FUNCTION "GCS7_SecCtrlMainMalting" : VOID	// FC 1060
TITLE = Section Control: Main function
//COPYRIGHT:    (C) 1994 BY  BUHLER AG,  CH-9240 UZWIL  SWITZERLAND
//
//PRODUCT:      GCS7
//
//TITLE:        SECTION CONTROL: MAIN PROGRAM
//
//-------------------------------------------------------------------------
//
//IDENT:        AUTOR:              DEPT:                         DATE:
//
//FC1060.1.0    M.Wedler            AEB31                         03-Feb-2005
//              Add. Code 1000 for Malting Plant only              
//FB60.3.5      A.Egli              CT3                           12-Nov-2003
//              Transition to Active: Set JobAc.BatchNo=1 when < 0
//FB60.3.4      A.Egli              CT3                           04-Aug-2003
//              PCRead.Status.StaImmediateStopASW is DBX120.0
//FB60.3.3      A.Egli              CT3                           17-Jul-2003
//              PCDirectControl: ParLineNr is DBW2 and not DBW4
//FB60.3.2      A.Egli              CT3                           12-Jun-2003
//              Wrong lenght copy Line to section
//FB60.3.1      A.Egli              CT3                           14-Mar-2003
//              Code35: Move to any section DB: DBW20=Destination
//              Code22,23: No Transition StEmptying to StWait
//FB60.3.0      A.Egli              CT3                            8-Okt-2002
//              New release
//FB60.2.10     A.Egli              CT3                           18-Mar-2002
//  Send Command only to next section, if InfDataReady=1
//FB60.2.9      A.Egli              CT3                           24-Sept-2001
//  ParStartReleaseTime <=0 : Unlimited time
//FB60.2.8      A.Egli              CT3                           17-Mai-2001
//  Update Last Batch in next section
//FB60.2.7      A.Egli              CT3                            5-Jul-2000
//  Read command from PC only with F_Define 
//FB60.2.6      A.Egli              CT3                           13-Mar-2000
//  Replace DBB73 with DBW72 and DBB9 with DBW8 
//FB60.2E       A.Egli              CT3                           30-Apr-1999
// -Zustandswechsel nach st_emptied: Abfrage DBX117.3 nicht DIX117.3 
//FB60.2D       A.Egli              CT3                           01-Apr-1999
// -Methode 25: Move allways
// -Bei reset Zustandswechsel nach st_emptied (Verbuchung
// -Bei reset kein Zustandswechsel nach  StActive
//FB60.2C       A.Egli              CT3                           22-Jul-98
//               Line-Nr =DBW2
//FB60.2B       A.Egli              AEE6                          14-Mai-98
//               ToASW.InfDataMoved
//FB60.2A       A.Egli              AEE6                          14-Jan-98
//               Update  S5 (Version 2M)
//FB60.1A       A.Egli              AEE6                          16-Jun-96
//               Convert S5 to S7 (Version 2H)
//
//-------------------------------------------------------------------------
//
//PURPOSE:      MANUAL : GCSOSMAN
//
//RESTRICTIONS:
//
//-------------------------------------------------------------------------
//
// CODE of the Methode
//        0    : METHODE CONTROL
//        1    : METHODE DECODER
//        2    : METHODE STEP
//        3    : METHODE STEP_TRANSITION
//        4    : METHODE STATE
//        5    : METHODE MOVE_DATA
//        6    : METHODE NEXT BATCH
//        7    : METHODE O_SECTION
//        9    : METHODE ResultTotal
//        10   : METHODE ResultBatch
//        12   : METHODE PC Direct Control (Diagnose)
//        13   : METHODE WayAdJustTime  
//        25   : METHODE MOVE_DATA Uncondtion
//        35   : METHODE MOVE_DATA any section
//
//ACTUAL DB BY CALL: SECTION  DB
//AUFGESCHALGENER  : SEKTIONS DB
//
//$EJECT
//
//
//
//
//
AUTHOR : EA
FAMILY : GCS7UL
NAME : SEC_MAIN
VERSION : 3.5
VAR_INPUT
  CODE : INT ;	// CODE
END_VAR
VAR_TEMP
  Fault : BOOL ;
  VarLength : INT ;
  tmpByteWrite : INT ;
  SecDBAc : INT ;
  SecDBNext : INT ;
END_VAR
BEGIN
NETWORK
TITLE =
      L     DBNO;
      T     #SecDBAc;
NETWORK
TITLE =  METHODE CONTROL
//Functions :
// - Section Commands 
//   > Sec.ToSSW.Func (commands last cycle) or'd with ToASW.Func
//   > Sec.ToASW.Func (commands) partially processed
// - Section Emptying Time controlled
// - Section F_Result controlled
//
//Called by : Section FC
      L     #CODE;
      L     0;	// METHODE CONTROL
      <>I;	// with Check JOB and Batch Status
      A(;
      L     #CODE;
      L     1000;	// METHODE CONTROL
      <>I;	// without Check JOB and Batch Status
      );
      JC    aEnd;
// === COMMANDS =====================================
      L     DBD 46;	// "SecDB".ToASW.Func
      L     DBD 66;	// "SecDB".ToSSW.Func
      OD;	// 
      T     DBD 46;	//>"SecDB".ToASW.Func
      L     0;	// 
      ==D;	// no new commands
      JC    aNoC;
// --- RESET STATUSBIT -----
      L     2#111111;	// ON-COMMAND
      L     DBW 46;	// "SecDB".ToASW.Func[31..16]
      AW;	// 
      INVI;	// 
      L     DBW 120;	// "SecDB".PCRead.Status[15..00]
      AW;	// 
      T     DBW 120;	//>"SecDB".PCRead.Status[15..00]
// --- SET STATUSBIT  ------
      L     2#11111111;	// OFF-COMMAND
      L     DBW 48;	// "SecDB".ToASW.Func[15..00]
      AW;	// 
      L     DBW 120;	// "SecDB".PCRead.Status[15..00]
      OW;	// 
      T     DBW 120;	//>"SecDB".PCRead.Status[15..00]
// 
// M.W. 03.02.05 
      L     #CODE;
      L     1000;	// METHODE CONTROL
      ==I;	// without Check JOB and Batch Status
      JC    nRes;
      JU    res;
nRes: NOP   0;
      R     DBX 48.1;	// "SecDB".ToASW.Func.CmdAbortBatch
      R     DBX 49.6;	// "SecDB".ToASW.Func.CmdReset
      R     DBX 49.7;	// "SecDB".ToASW.Func.CmdSequenzStop
//      R     DBX  121.0                  // "SecDB".PCRead.Status.StaImediateStop
      R     DBX 121.6;	// "SecDB".PCRead.Status.StaReset
      R     DBX 121.7;	//>"SecDB".PCRead.Status.StaEndOfJob
res:  NOP   0;
// 
      A     DBX 121.6;	// "SecDB".PCRead.Status.StaReset
      S     DBX 121.7;	//>"SecDB".PCRead.Status.StaEndOfJob
      A     DBX 48.1;	// "SecDB".ToASW.Func.CmdAbortBatch
      S     DBX 201.0;	//>"SecDB".JobAc.StaBatch.StaErrBatch
      A     DBX 49.6;	// "SecDB".ToASW.Func.CmdReset
      O     DBX 49.7;	// "SecDB".ToASW.Func.CmdSequenzStop
      O     DBX 48.1;	// "SecDB".ToASW.Func.CmdAbortBatch
      A     DBX 45.7;	// "SecDB".ToASW.InfDataReady [2.10]
      JCN   aNoC;
      CALL  "GCS7_SecCtrlSubMalting" (
           CODE                     := 2);	// SUBROUTINE sequenz_stop (Code 2)
aNoC: L     0;	// 
      T     DBD 66;	//>"SecDB".ToSSW.Func
      L     DBW 206;	// "SecDB".JobAc.BatchNo
      L     DBW 168;	// "SecDB".JobNom.BatchNo
      >=I;	// 
      S     DBX 201.3;	//>"SecDB".JobAc.StaBatch.StaLastBatch
// M.W.
      L     #CODE;
      L     1000;	// METHODE CONTROL
// M.W. 04.10.04
//      <>I                               // without Check JOB and Batch Status
      ==I;
      JC    aETI;	// -> Emptying Time
      CALL  "GCS7_SecCtrlSubMalting" (
           CODE                     := 1);	// SUBROUTINE compare (Code 1)
// === EMPTYING TIME ==================================
aETI: NOP   0;
      AN    DBX 64.2;	// "SecDB".ToSSW.InfPulseTimer
      O     DBX 45.0;	// "SecDB".ToASW.InfEmptyingTimeEnd
      JC    aE2;	// 
      L     DBW 132;	// "SecDB".PCRead.OutEmptyingTime
      +     1;	// 
      T     DBW 132;	//>"SecDB".PCRead.OutEmptyingTime
// 
aE2:  A     DBX 62.5;	// "SecDB".ToSSW.InfFeeding
      S     DBX 119.4;	//>"SecDB".PCRead.Status.StaLoaded
      A     DBX 64.7;	// "SecDB".ToSSW.InfReleaseEmptyingTime
      JC    aX3;	// 
      L     0;	// 
      T     DBW 132;	//>"SecDB".PCRead.OutEmptyingTime
aX3:  L     DBW 100;	// "SecDB".PCWrite.ParEmptyingTime
      L     DBW 132;	// "SecDB".PCRead.OutEmptyingTime
      <=I;	// 
      A     DBX 64.7;	// "SecDB".ToSSW.InfReleaseEmptyingTime 
      =     DBX 45.0;	// "SecDB".ToASW.InfEmptyingTimeEnd
      R     DBX 119.4;	//>"SecDB".PCRead.Status.StaLoaded
      AN    DBX 45.0;	// "SecDB".ToASW.InfEmptyingTimeEnd
      A     DBX 64.7;	// "SecDB".ToSSW.InfReleaseEmptyingTime
      =     DBX 119.6;	//>"SecDB".PCRead.Status.StaEmptyingTime
// === F_RESULT ========================================
      AN    DBX 64.1;	// "SecDB".ToSSW.CmdSendResult
      JC    aCMD;	// 
      AN    DBX 82.1;	// "SecDB".PCWrite.Hsk.Q_Result
      AN    DBX 201.2;	// "SecDB".JobAc.StaBatch.StaRegistrated
      AN    DBX 102.1;	// "SecDB".PCRead.Hsk.F_Result
      S     DBX 102.1;	//>"SecDB".PCRead.Hsk.F_Result
      S     DBX 41.0;	//>"SecDB".ChangeBit.CBit1 
aCMD: BEU;
aEnd: NOP   0;
NETWORK
TITLE =  METHODE DECODER (Code 1)
//Functions :
// -Copies Job data (obj64) from L_DB to all S_DB with the same job.
// -Calls initialise for sections with new job (F_Execute)
//
//Called by : Line FC
//Special : LCTRLMAIN INIT(1) must be called before this function
      L     #CODE;
      L     1;	// METHODE DECODER
      <>I;
      JC    bEnd;
      L     0;
      L     DBB 145;	// "LineDB".JobWrite.Hsk
      ==I;
      BEC;
      L     DBW 140;	// "LineDB".JobRead.ErrCode   [*1C*]
      L     0;
      <>I;
      BEC;
      L     64;	// Job Header
      T     DBW 20;	//>"LineDB".VarTemp[1] = ObjectNr
      CALL  FC 59 (
           $1                       := 1);	// SUBROUTINE Object Address (code 1)
      OPN   DI [DBW 4];	// >>> FIRST SECTION-DB[ "LineDB".Para.ParFirstSecDB]
bLop: AN    DIX 44.7;	// "SecDB".ToASW.InfSameJobLineDB
      JC    bNxt;
// === COMMANDS ========================================
      S     DIX 44.0;	//>"SecDB".ToASW.CmdModify  
      L     DBD 156;	// "LineDB".JobWrite.Func
      L     DID 46;	// "SecDB".ToASW.Func
      OD;	// 
      T     DID 46;	//>"SecDB".ToASW.Func
// === COPY JOB-HEADER (JObNom)=========================
      L     DINO;
      T     #SecDBAc;
      CALL  FC 49 (
           $1                       := P#DIX 4.0,
           $2                       := 160,
           $3                       := #SecDBAc,
           $4                       := 160,
           $5                       := 40,
           $6                       := #Fault);	// L_DB /  L_DB.JobNom /  S_DB /  S_DB.JobNom /  JobNom
// === COPY ADDITIONAL DATA (SecNom)====================
      L     DBW 22;	// "LineDB".VarTemp[2]= VarDWNr
      L     0;	// 
      ==I;	// 
      JC    bEXE;	// 
      L     DIW 12;	// "SecDB".Para.ParSecDataLenNomValue
      T     #VarLength;	//>VarLength
      L     DIW 10;	// "SecDB".Para.ParSecDataFirstByte
      L     DIW 14;	// "SecDB".Para.ParSecDataLenAcValue [3.1]
      +I;
      T     #tmpByteWrite;
      CALL  FC 49 (
           $1                       := P#DIX 4.0,
           $2                       := P#DBX 22.0,
           $3                       := #SecDBAc,
           $4                       := #tmpByteWrite,
           $5                       := #VarLength,
           $6                       := #Fault);	// L_DB /  L_DB.VarDWNr /  S_DB
bEXE: AN    DBX 145.1;	// "LineDB".JobWrite.Hsk.F_Execute
      JC    bNxt;
      R     DBX 153.7;	//>"LineDB".JobWrite.ObjMask[64]
      L     DBD 146;	// "LineDB".JobWrite.ObjMask[64..01]
      L     DBD 150;	// "LineDB".JobWrite.ObjMask[64..01]
      OD;
      JN    bNxt;
      CDB;
      CALL  "GCS7_SecCtrlSubMalting" (
           CODE                     := 3);	// SUBROUTINE init_section
      CDB;
// -- Call next section
bNxt: L     DIW 8;	// "SecDB".Para.ParNextSecDB
      L     0;	//  
      ==I;	// no next section
      JC    bINI;	// 
      OPN   DI [DIW 8];	//>>> NEXT SECTION-DB["SecDB".Para.ParNextSecDB]
      JU    bLop;
bINI: R     DBX 153.7;	//>"LineDB".JobWrite.ObjMask[64]
      BEU;
bEnd: NOP   0;
NETWORK
TITLE =  METHODE STEP (Code 2 , 22) 
//Functions :
// - Tests for step transitions from current step "SecDB".PCRead.Step
//   > Output SecDB".ToASW.Transition 
//
//Called by : Section FC
      L     #CODE;
      L     2;	// METHODE STEP
      <>I;
      A(;
      L     #CODE;
      L     22;
      <>I;
      );
      JC    cEnd;
      L     0;
      T     DBW 50;	// "SecDB".ToASW.Transition:=0
      A     DBX 111.0;	// "SecDB".PCRead.Step.StPassive
      JC    cS0;
      A     DBX 111.1;	// "SecDB".PCRead.Step.StWait
      JC    cS1;	// 
      A     DBX 111.2;	// "SecDB".PCRead.Step.StActive
      JC    cS2;
      A     DBX 111.3;	// "SecDB".PCRead.Step.StReady
      JC    cS3;
      A     DBX 111.4;	// "SecDB".PCRead.Step.StEmptying
      JC    cS4;
      A     DBX 111.5;	// "SecDB".PCRead.Step.StEmptied
      JC    cS5;
      A     DBX 111.6;	// "SecDB".PCRead.Step.StIdling
      JC    cS6;
      S     DBX 111.0;	// "SecDB".PCRead.Step.StPassive
// === "SecDB".PCRead.Step.StPassive ===================
cS0:  A     DBX 45.7;	// "SecDB".ToASW.InfDataReady
      JC    cTx1;	//>Transition.ToWait
      JU    cEnd;
// === "SecDB".PCRead.Step.StWait ======================
cS1:  A(;
      L     #CODE;
      L     2;
      ==I;
      );
      A     DBX 121.7;	// "SecDB".PCRead.Status.StaEndOfJob
      AN    DBX 44.5;	// "SecDB".ToASW.InfSameBatchPrevSec
      O     DBX 121.6;	// "SecDB".PCRead.Status.StaReset
      ON    DBX 45.7;	// "SecDB".ToASW.InfDataReady
      JC    cTx5;	//>Transition.ToEmptied [2D]
      AN    DBX 116.0;	// "SecDB".PCRead.fault.EsBatchSize
      A     DBX 63.1;	// "SecDB".ToSSW.CmdGotoActive
      JC    cTx2;	//>Transition.ToActive
      JU    cEnd;
// === "SecDB".PCRead.Step.StActive ====================
cS2:  A     DBX 63.2;	// "SecDB".ToSSW.CmdGotoReady
      AN    DBX 44.5;	// "SecDB".ToASW.InfSameBatchPrevSec
      JC    cTx3;	//>Transition.ToReady
      L     DBW 72;	// "SecDB".ToSSW.InNextSecDB
      L     0;	// 
      ==I;	// 
      O     DBX 44.6;	// "SecDB".ToASW.InfSameBatchNextSec
      AN    DBX 44.5;	// "SecDB".ToASW.InfSameBatchPrevSec
      A     DBX 63.3;	// "SecDB".ToSSW.CmdGotoEmptying
      JC    cTx4;	//>Transition.ToEmptying 
      A     DBX 121.6;	// "SecDB".PCRead.Status.StaReset
      ON    DBX 45.7;	// "SecDB".ToASW.InfDataReady
      JC    cTx5;	//>Transition.ToEmptied [2D]
      JU    cEnd;
// ===  "SecDB".PCRead.Step.StReady ====================
cS3:  L     DBW 72;	// "SecDB".ToSSW.InNextSecDB
      L     0;	// 
      ==I;	// 
      O     DBX 44.6;	// "SecDB".ToASW.InfSameBatchNextSec
      A     DBX 63.3;	// "SecDB".ToSSW.CmdGotoEmptying
      JC    cTx4;	//>Transition.ToEmptying 
      A     DBX 121.6;	// "SecDB".PCRead.Status.StaReset
      ON    DBX 45.7;	// "SecDB".ToASW.InfDataReady
      JC    cTx5;	//>Transition.ToEmptied [2D]
      JU    cEnd;
// === "SecDB".PCRead.Step.StEmptying ===================
cS4:  A     DBX 44.5;	// "SecDB".ToASW.InfSameBatchPrevSec
      JC    cTx2;	//>Transition.ToActive
      L     DBW 72;	// "SecDB".ToSSW.InNextSecDB
      L     0;	// 
      ==I;	// 
      O     DBX 44.6;	// "SecDB".ToASW.InfSameBatchNextSec
      A     DBX 63.4;	// "SecDB".ToSSW.CmdGotoEmptied
      JC    cTx5;	//>Transition.ToEmptied
      A     DBX 121.6;	// "SecDB".PCRead.Status.StaReset
      ON    DBX 45.7;	// "SecDB".ToASW.InfDataReady 
      JC    cTx5;	//>Transition.ToEmptied [2D]
      JU    cEnd;
// === "SecDB".PCRead.Step.StEmptied=====================
cS5:  A     DBX 44.5;	// "SecDB".ToASW.InfSameBatchPrevSec
      AN    DBX 121.6;	// "SecDB".PCRead.Status.StaReset [2D]
      JC    cTx2;	//>Transition.ToActive
      L     DBW 206;	// "SecDB".JobAc.BatchNo 
      L     DBW 168;	// "SecDB".JobNom.BatchNo
      >=I;	// 
      S     DBX 121.7;	//>"SecDB".PCRead.Status.StaEndOfJob
      L     0;	// 
      L     DBW 70;	// "SecDB".ToSSW.InPrevSecDB
      ==I;	// 
      A(;
      L     #CODE;
      L     22;
      <>I;
      );
      AN    DBX 121.6;	// "SecDB".PCRead.Status.StaReset 
      AN    DBX 121.7;	// "SecDB".PCRead.Status.StaEndOfJob
      A     DBX 45.7;	// "SecDB".ToASW.InfDataReady
      A     DBX 63.5;	// "SecDB".ToSSW.CmdGotoIdling
      JC    cTx1;	//>Transition.ToWait
      A     DBX 121.6;	// "SecDB".PCRead.Status.StaReset [2D]
      ON    DBX 45.7;	// "SecDB".ToASW.InfDataReady
      AN    DBX 119.3;	// "SecDB".PCRead.Status.StaOnline [2E]
      O     DBX 63.5;	// "SecDB".ToSSW.CmdGotoIdling
      JC    cTx6;	//>Transition.ToIdling
      JU    cEnd;
// === "SecDB".PCRead.Step.StIdling =====================
cS6:  A     DBX 45.7;	// "SecDB".ToASW.InfDataReady
      JC    cTx1;	//>Transition.ToWait
      A     DBX 63.6;	// "SecDB".ToSSW.CmdGotoPassive
      JC    cTx0;	//>Transition.ToPassive
      JU    cEnd;
// === SET TRANSITION ===================================
cTx0: L     2#1;	// "SecDB".ToASW.Transition.ToPassive
      JU    cTra;	// 
cTx1: L     2#10;	// "SecDB".ToASW.Transition.ToWait
      JU    cTra;	// 
cTx2: L     2#100;	// "SecDB".ToASW.Transition.ToActive
      JU    cTra;	// 
cTx3: L     2#1000;	// "SecDB".ToASW.Transition.ToReady
      JU    cTra;	// 
cTx4: L     2#10000;	// "SecDB".ToASW.Transition.ToEmptying
      JU    cTra;	// 
cTx5: L     2#100000;	// "SecDB".ToASW.Transition.ToEmptied
      JU    cTra;	// 
cTx6: L     2#1000000;	// "SecDB".ToASW.Transition.ToIdling
// ==== WRITE TRANSITION ================================
cTra: T     DBW 50;	//>"SecDB".ToASW.Transition
      BEU;
cEnd: NOP   0;
NETWORK
TITLE =  METHODE TRANSITION_STEP (code 3)
//Functions :
// - Manages Step Transitions "SecDB".ToASW.Transition
//   > Writes transition specific commands
//   > Output SecDB".ToASW.Step
//
//Called by : Section FC
      L     #CODE;
      L     3;	// METHODE TRANSITION STEP 
      <>I;
      A(;
      L     #CODE;
      L     23;
      <>I;
      );
      JC    dEnd;
      L     DBW 50;	// "SecDB".ToASW.Transition
      L     0;	// 
      ==I;	// 
      BEC;	// EXIT
      A     DBX 51.0;	// "SecDB".ToASW.Transition.ToPassive
      JC    dTx0;
      A     DBX 51.1;	// "SecDB".ToASW.Transition.ToWait
      JC    dTx1;
      A     DBX 51.2;	// "SecDB".ToASW.Transition.ToActive 
      JC    dTx2;
      A     DBX 51.3;	// "SecDB".ToASW.Transition.ToReady
      JC    dTx3;
      A     DBX 51.4;	// "SecDB".ToASW.Transition.ToEmptying
      JC    dTx4;
      A     DBX 51.5;	// "SecDB".ToASW.Transition.ToEmptied 
      JC    dTx5;
      A     DBX 51.6;	// "SecDB".ToASW.Transition.ToIdling
      JC    dTx6;
      JU    dEnd;
// === "SecDB".ToASW.Transition.ToPassive ===============
dTx0: NOP   0;
      JU    dTra;
// === "SecDB".ToASW.Transition.ToWait ==================
dTx1: R     DBX 63.1;	// "SecDB".ToSSW.CmdGotoActive 
      R     DBX 64.1;	// "SecDB".ToSSW.CmdSendResult
      A     DBX 111.5;	// "SecDB".PCRead.Step.StEmptied 
      R     DBX 201.0;	//>"SecDB".JobAc.StaBatch.StaErrBatch
      JU    dTra;
// === "SecDB".ToASW.Transition.ToActive ================
dTx2: R     DBX 63.2;	//>"SecDB".ToSSW.CmdGotoReady
      R     DBX 63.3;	//>"SecDB".ToSSW.CmdGotoEmptying
      R     DBX 64.1;	//>"SecDB".ToSSW.CmdSendResult
      L     DBW 206;	// "SecDB".JobAc.BatchNo  [3.5]
      L     1;	//                        [3.5]
      >=I;	//                        [3.5]
      ON    DBX 200.6;	// "SecDB".JobAc.StaBatch.StaEmptyingBatch [3.5]
      JC    dTra;	//                        [3.5]
      T     DBW 206;	// "SecDB".JobAc.BatchNo  [3.5]
      JU    dTra;
// === "SecDB".ToASW.Transition.ToReady =================
dTx3: R     DBX 63.3;	//>"SecDB".ToSSW.CmdGotoEmptying
      JU    dTra;
// === "SecDB".ToASW.Transition.ToEmptying ==============
dTx4: R     DBX 63.4;	//>"SecDB".ToSSW.CmdGotoEmptied
      JU    dTra;
// === "SecDB".ToASW.Transition.ToEmptied ===============
dTx5: R     DBX 63.5;	//>"SecDB".ToSSW.CmdGotoIdling
      JU    dTra;
// === "SecDB".ToASW.Transition.ToIdling ================
dTx6: R     DBX 63.6;	//>"SecDB".ToSSW.CmdGotoPassive
      R     DBX 201.0;	//>"SecDB".JobAc.StaBatch.StaErrBatch
      R     DBX 200.7;	//>"SecDB".JobAc.StaBatch.StaScaleRecipeValid
      AN    DBX 121.7;	// "SecDB".PCRead.Status.StaEndOfJob [2.8]
      JC    dT61;	// [2.8]                
      CALL  "GCS7_SecCtrlSubMalting" (
           CODE                     := 2);	// SUBROUTINE sequenz_stop [2.8]
dT61: L     0;	// 
      L     DBW 70;	// "SecDB".ToSSW.InPrevSecDB 
      <>I;	// 
      O(;
      L     #CODE;
      L     23;
      ==I;
      );
      O     DBX 121.7;	// "SecDB".PCRead.Status.StaEndOfJob
      R     DBX 45.7;	//>"SecDB".ToASW.InfDataReady
      CALL  "GCS7_SecCtrlSubMalting" (
           CODE                     := 7);	// Subroutine TestDone
      AN    DBX 39.0;	// OUTP.JobNotFound
      JC    dTra;	// 
      AN    DBX 102.0;	// "SecDB".PCRead.Hsk.F_Status 
      S     DBX 201.4;	//>"SecDB".JobAc.StaBatch.StaDone
      S     DBX 102.0;	//>"SecDB".PCRead.Hsk.F_Status
      S     DBX 41.0;	//>"SecDB".ChangeBit.CBit1
dTra: L     DBW 50;	// "SecDB".ToASW.Transition
      T     DBB 111;	//>"SecDB".PCRead.Step
      SET;	// 
      S     DBX 41.0;	//>"SecDB".ChangeBit.CBit1
      BEU;
dEnd: NOP   0;
NETWORK
TITLE =  METHODE STATE Code4
//Functions :
// - Processes SumState "SecDB".PCRead.State
//   > Output "SecDB".PCRead.State
//
//Called by : Section FC
      L     #CODE;
      L     4;	// METHODE STATE
      <>I;
      JC    eEnd;
      A     DBX 113.0;	// "SecDB".PCRead.State.StStopped
      JC    eS0;
      A     DBX 113.1;	// "SecDB".PCRead.State.StStarting
      JC    eS1;
      A     DBX 113.2;	// "SecDB".PCRead.State.StStarted 
      JC    eS2;
      A     DBX 113.3;	// "SecDB".PCRead.State.StStopping
      JC    eS3;
      A     DBX 113.5;	// "SecDB".PCRead.State.StFeeding
      JC    eS4;
      S     DBX 113.0;	// "SecDB".PCRead.State.StStopped
// === "SecDB".PCRead.State.StStopped ===================
eS0:  AN    DBX 62.0;	// "SecDB".ToSSW.InfStopped
      JC    eT01;	//>State.StStarting
      JU    eEnd;	// 
eT01: L     2#10;	//>"SecDB".PCRead.State.StStarting
      JU    eTra;
// === "SecDB".PCRead.State.StStarting ==================
eS1:  A     DBX 62.2;	// "SecDB".ToSSW.InfStarted
      JC    eT12;	//>State.StStarted
      A     DBX 120.0;	// "SecDB".PCRead.Status.StaImmediateStopASW // [3.4]
      O     DBX 62.0;	// "SecDB".ToSSW.InfStopped
      O     DBX 111.6;	// "SecDB".PCRead.Step.StIdling
      JC    eT13;	//>State.StStopping
      JU    eEnd;
eT12: L     2#100;	//>"SecDB".PCRead.State.StStarted
      JU    eTra;
eT13: L     2#1000;	//>"SecDB".PCRead.State.StStopping
      JU    eTra;
// === "SecDB".PCRead.State.StStarted ===================
eS2:  A     DBX 120.0;	// "SecDB".PCRead.Status.StaImmediateStopASW
      O     DBX 62.0;	// "SecDB".ToSSW.InfStopped
      JC    eT23;	//>State.StStopping
      AN    DBX 62.2;	// "SecDB".ToSSW.InfStarted
      JC    eT21;	//>State.StStarting
      A     DBX 62.5;	// "SecDB".ToSSW.InfFeeding
      JC    eT25;	//>State.StFeeding
      JU    eEnd;
eT21: L     2#10;	//>"SecDB".PCRead.State.StStarting
      JU    eTra;
eT23: L     2#1000;	//>"SecDB".PCRead.State.StStopping
      JU    eTra;
eT25: L     2#100000;	//>"SecDB".PCRead.State.StFeeding
      JU    eTra;
// === "SecDB".PCRead.State.StStopping ==================
eS3:  A     DBX 62.0;	// "SecDB".ToSSW.InfStopped
      JC    eT30;	//>State.StStopped
      AN    DBX 120.0;	// "SecDB".PCRead.Status.StaImmediateStopASW
      AN    DBX 62.0;	// "SecDB".ToSSW.InfStopped
      A     DBX 62.2;	// "SecDB".ToSSW.InfStarted
      JC    eT32;	//>State.StStarted
      AN    DBX 120.0;	// "SecDB".PCRead.Status.StaImmediateStopASW
      AN    DBX 111.6;	// "SecDB".PCRead.Step.StIdling
      JC    eT32;	//>State.StStarting
      JU    eEnd;
eT30: L     2#1;	//>"SecDB".PCRead.State.StStopped
      JU    eTra;
eT32: L     2#100;	//>"SecDB".PCRead.State.StStarted
      JU    eTra;
      L     2#10;	//>"SecDB".PCRead.State.StStarting
      JU    eTra;
// === "SecDB".PCRead.State.StFeeding ===================
eS4:  AN    DBX 62.5;	// "SecDB".ToSSW.InfFeeding
      JC    eT52;	//>State.StStarted
      JU    eEnd;	// 
eT52: L     2#100;	//>"SecDB".PCRead.State.StStarted
// ==== SET STATE (TRANSITION) ==========================
eTra: T     DBB 113;	//>"SecDB".PCRead.State
      SET;	// 
      S     DBX 41.0;	//>"SecDB".Changebit.CBit1
      BEU;
eEnd: NOP   0;
NETWORK
TITLE =  METHODE MOVE_DATA Code 5,25,35
//Function :
// - Manages Section to Section Job Copy for Job and Bin Data 
// > Code 5: Regular copy to next section
// > Code 25:Unconditional copy to next section
// > Code 35:Regular copy to specified section destination (DBW20)
// > Output : Job Ac, Job Nom, Sec Ac, Sec Nom, Bin Recipe. Copied Section to 
//Section 
//
//Called by : Section FC
      L     #CODE;
      L     5;	// METHODE MOVE DATA Next Section Regular
      ==I;
      JC    m5;
      L     #CODE;
      L     25;	// METHODE MOVE DATA Next Section Unconditional
      ==I;
      JC    m25;
      L     #CODE;
      L     35;	// METHODE MOVE DATA Any Section Regular
      <>I;
      JC    fEnd;
// === Move to section DBW20 (Code 35)===============
      R     DBX 44.2;	// S_DB[n  ].ToASW.CmdDataMoved
      L     0;
      L     DBW 20;	// S_DB[n  ].VarTemp.InOutValue1
      ==I;	// 
      BEC;	//>No next section
      T     #SecDBNext;
      OPN   DI [#SecDBNext];	// >>>CALL NEXT SECTION ["SecDB".ToSSW.InNextSecDB]
      JU    m35;	//> Regular Conditions
//====== Move Uncondition (Code=25) =================
m25:  R     DBX 44.2;	// S_DB[n  ].ToASW.CmdDataMoved
      L     DBW 72;	// S_DB[n  ].ToSSW.InNextSecDB
      L     0;	// 
      ==I;	// 
      BEC;	//>No next section
      AN    DBX 44.6;	// S_DB[n  ].ToASW.InfSameBatchNextSec
      OPN   DI [DBW 72];	// >>> NEXT SECTION ["SecDB".ToSSW.InNextSecDB]
      A     DIX 64.0;	// S_DB[n+1].ToSSW.InfReadyForNewBatch
      AN    DIX 121.3;	// S_DB[n+1].PCRead.Status.StaHold
      A(;
      AN    DIX 102.0;	// S_DB[n+1].PCRead.Hsk.F_Status
      ON    DIX 119.3;	// S_DB[n+1].PCRead.Status.StaOnline
      );
      JC    C3;	//>Move Data
      BEU;
//=== Move Regular (Code=5) =========================
m5:   R     DBX 44.2;	// S_DB[n  ].ToASW.CmdDataMoved
      A     DBX 44.6;	// S_DB[n  ].ToASW.InfSameBatchNextSec
      BEC;	//  
      L     DBW 72;	// S_DB[n  ].ToSSW.InNextSecDB
      L     0;	// 
      ==I;	// 
      BEC;	//>No next section
      OPN   DI [DBW 72];	// >>> NEXT SECTION-DB["SecDB".ToSSW.InNextSecDB]
m35:  A     DBX 201.0;	// S_DB[n  ].JobAc.StaBatch.StaErrBatch
      A     DIX 45.7;	// S_DB[n+1].ToASW.InfDataReady
      BEC;	// 
      A     DIX 165.0;	// S_DB[n+1].sta_err_batch
      A     DIX 45.7;	// S_DB[n+1].ToASW.InfDataReady
      BEC;	// 
      A     DIX 111.0;	// S_DB[n+1].PCRead.Step.StPassive
      O     DIX 111.6;	// S_DB[n+1].PCRead.Step.StIdling
      O     DIX 111.4;	// S_DB[n+1].PCRead.Step.StEmptying
      O     DIX 111.5;	// S_DB[n+1].PCRead.Step.StEmptied
      JC    C2;
      BEU;
      AN    DBX 45.7;	// S_DB[n  ].ToASW.InfDataReady
      O     DBX 44.3;	// S_DB[n  ].ToASW.InfSameJobPrevSec
      A     DBX 64.0;	// S_DB[n  ].ToSSW.InfReadyForNewBatch
      AN    DBX 121.3;	// S_DB[n  ].PCRead.Status.StaHold
      A(;
      AN    DBX 102.0;	// S_DB[n  ].PCRead.Hsk.F_Status
      ON    DBX 119.3;	// S_DB[n  ].PCRead.Status.StaOnline
      );
C2:   AN    DIX 45.7;	// S_DB[n+1].ToASW.InfDataReady
      O     DIX 44.3;	// S_DB[n+1].ToASW.InfSameJobPrevSec
      A     DIX 64.0;	// S_DB[n+1].ToSSW.InfReadyForNewBatch
      AN    DIX 121.3;	// S_DB[n+1].PCRead.Status.StaHold
      A(;
      AN    DIX 102.0;	// S_DB[n+1].PCRead.Hsk.F_Status
      ON    DIX 119.3;	// S_DB[n+1].PCRead.Status.StaOnline
      );
      JC    C3;
      BEU;
// === MOVE DATA =======================================
// --- Copy Header (JobAc + JobNom)---------------------
C3:   L     DINO;
      T     #SecDBNext;
      CALL  FC 49 (
           $1                       := #SecDBAc,
           $2                       := 160,
           $3                       := #SecDBNext,
           $4                       := 160,
           $5                       := 80,
           $6                       := #Fault);	// S_DB[n  ].JobNom /  S_DB[n+1].JobNom /  JobAc + JobNom
// --- Copy Dynamic Datas (SecAc + SecNom)--------------
      L     DIW 14;	// S_DB[n+1].Para.ParSecDataLenAcValue
      L     DIW 12;	// S_DB[n+1].Para.ParSecDataLenNomValue
      +I;
      T     #VarLength;
      CALL  FC 49 (
           $1                       := #SecDBAc,
           $2                       := P#DBX 10.0,
           $3                       := #SecDBNext,
           $4                       := P#DIX 10.0,
           $5                       := #VarLength,
           $6                       := #Fault);	// S_DB[n  ].Para.ParSecDataFirstByte /  S_DB[n+1].Para.ParSecDataFirstByte /  SecAc + SecNom
// --- Copy Bin Data (Recipe) ---------------------------
      CALL  FC 49 (
           $1                       := #SecDBAc,
           $2                       := P#DBX 16.0,
           $3                       := #SecDBNext,
           $4                       := P#DIX 16.0,
           $5                       := P#DIX 18.0,
           $6                       := #Fault);	// S_DB[n  ].Para.ParBinDataFirstByte /  S_DB[n+1].Para.ParBinDataFirstByte /  S_DB[n+1].Para.ParBinDataLength
// --- Initalise S_DB[n+1] ------------------------------
      SET;
      S     DIX 45.7;	// S_DB[n+1].ToASW.InfDataReady 
      S     DIX 44.1;	// S_DB[n+1].ToASW.CmdNewBatch
      S     DBX 44.2;	// S_DB[n  ].ToASW.CmdDataMoved
      R     DIX 121.6;	// S_DB[n+1].PCRead.Status.StaReset
      R     DIX 121.7;	// S_DB[n+1].PCRead.Status.StaEndOfJob
      R     DIX 64.1;	// S_DB[n+1].ToSSW.CmdSendResult
      AN    DBX 121.0;	// S_DB[n  ].PCRead.Status.StaImmediateStop   
      R     DIX 121.0;	// S_DB[n+1].PCRead.Status.StaImmediateStop      
      AN    DBX 121.1;	// S_DB[n  ].PCRead.Status.StaTransferOff
      R     DIX 121.1;	// S_DB[n+1].PCRead.Status.StaTransferOff
      AN    DBX 121.2;	// S_DB[n  ].PCRead.Status.StaFeedOff
      R     DIX 121.2;	// S_DB[n+1].PCRead.Status.StaFeedOff
      CDB;	// >>> DB to DI
      CALL  "GCS7_SecCtrlSubMalting" (
           CODE                     := 1);	//SUBROUTINE compare S_DB[n+1]
      CDB;	// >>> DB to DI
      CALL  "GCS7_SecCtrlSubMalting" (
           CODE                     := 1);	//SUBROUTINE compare S_DB[n  ]
      BEU;
fEnd: NOP   0;
NETWORK
TITLE =  METHODE NEXT_BATCH (code 6)
//Function : 
//  - Batch change functions
//    > "SecDB".JobAc.BatchNo Incremented
//    > "SecDB".JobAc.BatchWeightTarget Calculated 
//    > Batch change commands set
//
//Called by : Section FC in Batch Mixing Applications
      L     #CODE;
      L     6;	// METHODE NEXT BATCH
      <>I;
      JC    gEnd;
      L     DBW 206;	// "SecDB".JobAc.BatchNo
      L     DBW 188;	// "SecDB".JobNom.BatchNoOffset
      >=I;
      JC    gOK;
      T     DBW 206;	//>"SecDB".JobAc.BatchNo
gOK:  A     DBX 121.7;	// "SecDB".PCRead.Status.StaEndOfJob
      BEC;	// 
// === START BATCH =====================================
      CALL  "GCS7_SecCtrlSubMalting" (
           CODE                     := 6);	// Subroutine CalcBatchSize
      A     DBX 116.0;	// "SecDB".PCRead.Fault.EsBatchSize
      O     DBX 121.7;	// "SecDB".PCRead.Status.StaEndOfJob
      BEC;
      L     DBD 210;	// "SecDB".JobAc.BatchWeightTarget
      L     DBD 202;	// "SecDB".JobAc.JobWeight
      +D;	// 
      T     DBD 202;	//>"SecDB".JobAc.JobWeight
      L     DBW 206;	// "SecDB".JobAc.BatchNo
      +     1;	// 
      T     DBW 206;	//>"SecDB".JobAc.BatchNo
      L     0;
      T     DBD 214;	//>"SecDB".JobAc.BatchWeightActual
      SET;
      R     DBX 201.1;	//>"SecDB".JobAc.StaBatch.StaHandAddReady
      R     DBX 201.2;	//>"SecDB".JobAc.StaBatch.StaRegistrated
      L     DBW 206;	// "SecDB".JobAc.BatchNo
      L     DBW 168;	// "SecDB".JobNom.BatchNo
      >=I;	// 
      S     DBX 201.3;	//>"SecDB".JobAc.StaBatch.StaLastBatch 
      SET;	// 
      S     DBX 45.7;	//>"SecDB".ToASW.InfDataReady
      S     DBX 44.1;	//>"SecDB".ToASW.CmdNewBatch
      CALL  "GCS7_SecCtrlSubMalting" (
           CODE                     := 1);	// SUBROUTINE compare S_DB[n]
      BEU;
gEnd: NOP   0;
NETWORK
TITLE =  METHODE O_SECTION (Code 7)
//Function :
// - "SecDB".PCWrite.Func Or'd with "SecDB".ToASW.Func on PCWrite.Hsk.F_Define
// - "SecDB".PCWrite.Hsk. processed
//
//Called by : Section FC
      L     #CODE;
      L     7;	//METHODE O_SECTION
      <>I;
      JC    hEnd;
      L     DBW 82;	// "SecDB".PCWrite.Hsk
      L     0;
      ==I;
      BEC;
// === COMMANDS ========================================
      AN    DBX 83.0;	// "SecDB".PCWrite.Hsk.F_Define [2.7]
      JC    hDef;	// 
      L     DBD 46;	// "SecDB".ToASW.Func
      L     DBD 86;	// "SecDB".PCWrite.Func
      OD;	// 
      T     DBD 46;	//>"SecDB".ToASW.Func
// === Q_RESULT ========================================
hDef: AN    DBX 82.1;	// "SecDB".PCWrite.Hsk.Q_Result
      JC    hIni;
      S     DBX 201.2;	//>"SecDB".JobAc.StaBatch.StaRegistrated 
// === INIT INTERFACE ==================================
hIni: L     DBB 82;	// "SecDB".PCWrite.Hsk.Q_xxxx
      INVI;
      L     DBB 102;	// "SecDB".PCRead.Hsk.F_
      AW;	// Reset Cleared HS
      T     DBB 102;	//>"SecDB".PCRead.Hsk.F_xxxx
      L     0;
      T     DBW 82;	//>"SecDB".PCWrite.Hsk
      SET;
      S     DBX 41.1;	//>"SecDB".ChangeBit.CBit2
      BEU;
hEnd: NOP   0;
NETWORK
TITLE =  METHODE ResultTotal (Code=9)
//Function : 
// - Adds Weight DBD32 into all Sections with Same Job Number
//output : S_DB.JobAc.JobWeight  
//
//Called by : Scale Management or ASW
      L     #CODE;
      L     9;	// METHODE RESULT TOTAL
      <>I;
      JC    iEnd;
      OPN   DI [DBW 4];	//>>> LINE DI["L_DB".Para.ParLineDB]
      OPN   DI [DIW 4];	//>>> FIRST SEC DI["S_DB".Para.ParFirstSecDB]
//Loop over all section
iLop: AN    DIX 45.7;	// S_DI.ToASW.InfDataReady
      JC    iNxt;
      L     DID 160;	// S_DI.JobNom.JobNr
      L     DBD 160;	// S_DB.JobNom.JobNr
      <>D;	// 
      JC    iNxt;
      L     DBD 32;	// S_DB.VarTemp.InOutValue5 (Input value for registration)
      L     DID 202;	// S_DI.JobAc.JobWeight
      +D;	// 
      T     DID 202;	//>S_DI.JobAc.JobWeight
iNxt: L     0;	// 
      L     DIW 8;	// S_DI.Para.ParNextSecDB
      ==I;	// no further sections
      BEC;	// 
      OPN   DI [DIW 8];	//>>> NEXT SEC DI["SecDB".Para.ParNextSecDB]
      JU    iLop;
iEnd: NOP   0;
NETWORK
TITLE =  METHODE TotalBatch (Code=10)
//Function : 
// - Adds Weight DBD32 into all Sections with Same Batch
//output : S_DB.JobAc.BatchWeightActual  
//
//Called by : Scale Management or ASW
      L     #CODE;
      L     10;	// METHODE RESULT BATCH
      <>I;
      JC    jEnd;
      OPN   DI [DBW 4];	//>>> LINE DI["SecDB".Para.ParLineDB]
      OPN   DI [DIW 4];	//>>> FIRST SEC DI["LineDB".Para.ParFirstSecDB]
//Loop over all section
jLop: AN    DIX 45.7;	// S_DI.ToASW.InfDataReady
      JC    jNxt;
      L     DID 160;	// S_DI.JobNom.JobNr
      L     DBD 160;	// S_DB.JobNom.JobNr
      <>D;	//  
      JC    jNxt;
      L     DIW 206;	// S_DI.JobAc.BatchNo
      L     DBW 206;	// S_DB.JobAc.BatchNo
      <>I;	//  
      JC    jNxt;
      L     DBD 32;	// S_DB.VarTemp.InOutValue  Input value for registration
      L     DID 214;	// S_DI.JobAc.BatchWeightActual
      +D;	//  
      T     DID 214;	//>S_DI.JobAc.BatchWeightActual
jNxt: L     0;	// 
      L     DIW 8;	// S_DI.Para.ParNextSecDB
      ==I;	// 
      BEC;	// 
      OPN   DI [DIW 8];	//>>> NEXT SEC DI["SecDB".Para.ParNextSecDB]
      JU    jLop;
jEnd: NOP   0;
NETWORK
TITLE =  PC Direct Control (Diagnose) (code= 12)
//Function : 
//- Operate Direct Control Interface to Section
//
//Called by : Line FC
      L     #CODE;
      L     12;	// PC DIRECT CONTROL
      <>I;
      JC    kEnd;
      OPN   DI 3;
      L     0;
      L     DIW 42;	// DB3.PC.Hsk
      ==I;	// 
      BEC;	// 
//-- TEST OBJECT ---------------------------------------
      L     DIW 48;	// DB3.PC.ObjectType
      L     4000;
      <>I;
      BEC;
      L     DIW 50;	// DB3.PC.ObjectNo
      SRW   8;
      L     DBW 2;	// "SecDB".Para.ParLineDB [3.3]
      <>I;
      BEC;
      L     DIB 51;	// DB3.PC.ObjectNo (low byte)
      T     DBW 20;	//>"SecDB".VarTemp[1] ==VarSecNr
      CALL  "GCS7_SecCtrlSubMalting" (
           CODE                     := 4);	// SUBROUTINE SearchSection
      L     0;
      T     DBW 22;	//>"SecDB".VarTemp[2] == Search_mode=SectionNr
      CALL  "GCS7_SecCtrlSubMalting" (
           CODE                     := 4);	// SUBROUTINE SearchSection
      L     DBW 22;	// "SecDB".VarTemp[2]
      L     0;
      ==I;
      L     20;	// Error code: illegal_object
      JC    ERRO;	//>illegal section-nr
// --- PROCESS OBJECT ----------------------------------
      OPN   DB [DBW 22];	// CALL DB["SecDB".VarTemp[2]] = VarSecDB
// --- COMMANDS ----------------------------------------
      AN    DIX 43.0;	// DB3.PC.Hsk.FDefineCmd
      JC    D2;	// 
      L     DID 52;	// DB3..PC.Cmd1
      L     DBD 46;	// "SecDB".ToASW.Func
      OD;	// 
      T     DBD 46;	//>"SecDB".ToASW.Func
// --- PARAMETERS --------------------------------------
D2:   AN    DIX 43.1;	// DB3.PC.Hsk.FDefineCmd
      JC    EXAM;	// 
      L     DIW 58;	// DB3.PC.Value[1]
      T     DBW 90;	//>"SecDB".PCWrite.Value1
      L     DIW 60;	// DB3.PC.Value[2]
      T     DBW 92;	//>"SecDB".PCWrite.Value2
      L     DIW 62;	// DB3.PC.Value[3]
      T     DBW 94;	//>"SecDB".PCWrite.Value3
      L     DIW 64;	// DB3.PC.Value[4]
      T     DBW 96;	//>"SecDB".PCWrite.ParWayAdjustTime
      L     DIW 66;	// DB3.PC.Value[5]
      T     DBW 98;	//>"SecDB".PCWrite.Value5
      L     DIW 68;	// DB3.PC.Value[6]
      T     DBW 100;	//>"SecDB".PCWrite.ParEmptyingTime
// --- EXAMINE ------------------------------------------
EXAM: AN    DIX 43.3;	// DB3.PC.Hsk.FExamine
      JC    DONE;	// 
      L     DBD 90;	// 
      T     DID 58;	//>DB3.Value[1..2]
      L     DBD 94;	// 
      T     DID 62;	//>DB3.Value[3..4]
      L     DBD 98;	// 
      T     DID 66;	//>DB3.Value[5..6]
DONE: L     0;
ERRO: T     DB3.DBW 46;	//>DB3.PC.ErrCode
      L     0;	// 
      T     DB3.DBW 42;	//>DB3.PC.Hsk
      SET;	//  
      S     DB3.DBX 41.0;	//>DB3.ChangeBit.CBit1
      BEU;
kEnd: NOP   0;
NETWORK
TITLE = Methode WayAdJsutTime
//Function : 
// - Controls the Section Way Adjust Time to run from ToASW.CmdNewWay
// > Output : "SecDB".PCRead.OutWayAdjustTime
//
//Called by : Section FC
      L     #CODE;
      L     13;	// METHODE WAY ADJUST TIME
      <>I;
      JC    lEnd;
      AN    DBX 64.3;	// "SecDB".ToSSW.CmdNewWay
      JC    lJ1;
      R     DBX 45.1;	//>"SecDB".ToASW.InfWayAdjustTimeEnd
      R     DBX 64.3;	//>"SecDB".ToSSW.CmdNewWay
      L     0;
      T     DBW 128;	//>"SecDB".PCRead.OutWayAdjustTime
lJ1:  A     DBX 45.1;	// "SecDB".ToASW.InfWayAdjustTimeEnd
      BEC;
      AN    M 10.3;
      BEC;
      L     DBW 128;	// "SecDB".PCRead.OutWayAdjustTime
      +     2;
      T     DBW 128;	//>"SecDB".PCRead.OutWayAdjustTime
      L     DBW 96;	// "SecDB".PCWrite.ParWayAdjustTime
      >=I;
      S     DBX 45.1;	//>"SecDB".ToASW.InfWayAdjustTimeEnd
      BEU;
lEnd: NOP   0;
END_FUNCTION

FUNCTION "GCS7_SecCtrlSubMalting" : VOID	// FC 1061
TITLE = Section Control: Subroutines
//COPYRIGHT:    (C) 1994 BY  BUHLER LTD.
//                           CH-9240 UZWIL  SWITZERLAND
//
//PRODUCT:      GCS7
//
//TITLE:        SECTION CONTROL: SUBROUTINE
//
//-------------------------------------------------------------------------
//
//IDENT:        AUTOR:              DEPT:                         DATE:
//
//FB61.2.2      M.Wedler            AEB31                         31-Aug-2004
//             InfNextSectionFeeding   
//FB61.2.1      A.Egli              CT3                           12-Aug-2003
//              - Compare Prev Section
//FB61.2.0      A.Egli              CT3                            8-Okt-2002
//              - New release
//              - ToASW.InfSameBatchAnyPrevSec 
//              - ToASW.IntSameJobAnyPrevSec 
//FB61.1.5      A.Egli              CT3                            3-Jan-2002
//              Test minimum size : test < not <=
//FB61.1.4      A.Egli              CT3                           14-Apr-2000
//              Test Job active
//FB61.1D       A.Egli              CT3                           11-Juni-1999
//              Calculate number of batch: RND+
//FB61.1C       A.Egli              CT3                           20-Apr-1999
//              Reset EsBatchSizeUpdate by InitSection
//FB61.1B       A.Egli              AEE61                         14-Jan-98
//              Update  to S5 (Version 2G)
//FB61.1A       A.Egli              AEE61                         20-Jun-96
//              Convert to S7 (Version 2F)
//
//-------------------------------------------------------------------------
//
//PURPOSE:      MANUAL : GCSOSMAN
//
//RESTRICTIONS:
//
//-------------------------------------------------------------------------
//
//PARAMETER:
//---------
//  CODE: CODE of the Subroutine
//        KF +1    : SUBROUTINE TEST_MATERIAL
//        KF +2    : SUBROUTINE SEQUENZ_STOP
//        KF +3    : SUBROUTINE INIT_SECTION
//        KF +4    : SUBROUTINE SEARCH_SECTION
//        KF +5    : SUBROUTINE SEARCH_JOB
//        KF +6    : SUBROUTINE CALC_BATCH_SIZE
//        KF +7    : SUBROUTINE TestDone
//
//
AUTHOR : EA
FAMILY : GCS7UL
NAME : SEC_SUBR
VERSION : 2.1
VAR_INPUT
  CODE : INT ;	// CODE
END_VAR
VAR_TEMP
  VarLoop2 : BOOL ;
  VarLastBatch : INT ;
  VarRest : DINT ;
  tmpSameJob : BOOL ;
  tmpSameBatch : BOOL ;
END_VAR
BEGIN
NETWORK
TITLE =
NETWORK
TITLE =  COMPARE (Code 1)
//FLAG IN SUBROUTINE COMPARE: (Batch in previous section and next section)
//==========================
//
      L     #CODE;
      L     1;
      <>I;
      JC    aEND;
      R     DBX 44.3;	// S[n].ToASW.InfSameJobPrevSec
      R     DBX 44.5;	// S[n].ToASW.InfSameBatchPrevSec
      R     DBX 45.2;	// S[n].ToASW.InfSameJobAnyPrevSec
      R     DBX 45.3;	// S[n].ToASW.InfSameBatchAnyPrevSec
      OPN   DI [DBW 4];	//>>Call LineDB  DI["SecDB".Para.ParLineDB]
      OPN   DI [DIW 4];	//>>Call SecDB   DI["LineDB".Para.ParFirstSecDB]
//============================================
//Loop Prev sections
//============================================
pLop: L     DINO;	//Prev Section DB 
      L     DBNO;	//Actual Section DB
      ==I;
      JC    aNXT;
//-- Compare prev. Section
      L     DID 160;	// S[n-1].JobNom.JobNr
      L     DBD 160;	// S[n  ].JobNom.JobNr
      ==D;	// 
      A     DIX 45.7;	// S[n-1].ToASW.InfDataReady
      A     DBX 45.7;	// S[n].ToASW.InfDataReady  [2.1]
      AN    DIX 111.1;	// S[n-1].PCRead.Step.StWait
      =     #tmpSameJob;
      S     DBX 45.2;	// ->S[n].ToASW.InfSameJobAnyPrevSec
      L     DINO;	// Prev Section DB 
      L     DBW 70;	// "SecDB".ToSSW.InPrevSecDB
      ==I;
      A     #tmpSameJob;
      S     DBX 44.3;	// ->S[n].ToASW.InfSameJobPrevSec
//Compare batch
      L     DIW 206;	// S[n-1].JobAc.BatchNo
      L     DBW 206;	// S[n].JobAc.BatchNo
      ==I;	// 
      A     #tmpSameJob;
      =     #tmpSameBatch;
      S     DBX 45.3;	// S[n].ToASW.InfSameBatchAnyPrevSec
      L     DINO;	// Prev Section DB 
      L     DBW 70;	// "SecDB".ToSSW.InPrevSecDB
      ==I;
      A     #tmpSameBatch;
      S     DBX 44.5;	//  )->S[n].ToASW.InfSameBatchPrevSec
//Next 
      L     0;
      L     DIW 8;	// S[i].Para.ParNextSecDB
      ==I;
      JC    aNXT;
      OPN   DI [DIW 8];	//-->  Call next SecDB  DI[Para.ParNextSecDB]
      JU    pLop;
//End Loop Prev sections
//============================================
// Compare next Section
//============================================
aNXT: L     DBW 72;	// "SecDB".ToSSW.InNextSecDB
      L     0;	// 
      <>I;	// 
      A     DBX 45.7;	// "SecDB".ToASW.InfDataReady
      JC    aCM2;	// 
      R     DBX 44.4;	//"SecDB".ToASW.InfSameJobNextSec
      R     DBX 44.6;	//"SecDB".ToASW.InfSameBatchNextSec
      BEU;
aCM2: OPN   DI [DBW 72];	// -> CALL NEXT SECTION DB["SecDB".ToSSW.InNextSecDB]
      L     DID 160;	// S[n+1].JobNom.JobNr
      L     DBD 160;	// "SecDB".JobNom.JobNr
      ==D;
      A     DIX 45.7;	// S[n+1].ToASW.InfDataReady
      AN    DBX 111.1;	// "SecDB".PCRead.Step.StWait
      =     DBX 44.4;	// ->"SecDB".ToASW.InfSameJobNextSec
      L     DIW 206;	// S[n+1].JobAc.BatchNo
      L     DBW 206;	// "SecDB".JobAc.BatchNo
      ==I;
      A     DBX 44.4;	// "SecDB".ToASW.InfSameJobNextSec
      =     DBX 44.6;	// ->S"SecDB".ToASW.InfSameBatchNextSec
// M.W.                                
      A     DBX 44.4;	// "SecDB".ToASW.InfSameJobNextSec
      A     DBX 44.6;	// "SecDB".ToASW.InfSameBatchNextSec
      A     DIX 62.5;	// S[n+1].ToSSW.InfFeeding
      =     DBX 45.4;	// ->S"SecDB".ToASW.InfNextSectionFeeding
      BEU;
aEND: NOP   0;
NETWORK
TITLE =  SEQUENZ_STOP
//1.Scan : Serach last batch
//2.Scan : Set Bit last batch
      L     #CODE;
      L     2;
      <>I;
      JC    bEnd;
      R     #VarLoop2;
      L     0;
      T     #VarLastBatch;
bLo2: OPN   DI [DBW 4];	//>>Call LineDB  DI["SecDB".Para.ParLineDB]
      OPN   DI [DIW 4];	//>>Call SecDB   DI["LineDB".Para.ParFirstSecDB]
//Loop over all section
bLop: L     DID 160;	// S[i].JobNom.JobNr
      L     DBD 160;	// "SecDB".JobNom.JobNr
      <>D;	// 
      JC    bNEQ;	// 
      AN    #VarLoop2;
      JC    bL1;
// ==== LOOP2 =====================
      L     DIW 206;	// S[i].JobAc.BatchNo
      L     #VarLastBatch;
      ==I;	// 
      A     DBX 121.7;	// "SecDB".PCRead.Status.StaEndOfJob
      S     DIX 201.3;	// -> S[i].JobAc.StaBatch.StaLastBatch
      JU    bNEQ;
// === LOOP 1 =====================
bL1:  A     DBX 121.7;	// "SecDB".PCRead.Status.StaEndOfJob 
      S     DIX 121.7;	// ->S[i].PCRead.Status.StaEndOfJob
      L     #VarLastBatch;
      L     DIW 206;	// S[i].JobAc.BatchNo
      >=I;
      JC    bJ1;
      T     #VarLastBatch;
bJ1:  L     DIW 206;	// S[i].JobAc.BatchNo
      L     DBW 206;	// "SecDB".JobAc.BatchNo
      ==I;
      A     DBX 201.0;	// "SecDB".JobAc.StaBatch.StaErrBatch
      S     DIX 201.0;	// ->S[i].JobAc.StaBatch.StaErrBatch
bNEQ: L     0;
      L     DIW 8;	// S[i].Para.ParNextSecDB
      ==I;
      JC    bL2;
      OPN   DI [DIW 8];	//-->  Call next SecDB  DI[Para.ParNextSecDB]
      JU    bLop;
//2nd Loop
bL2:  A     #VarLoop2;
      BEC;
      S     #VarLoop2;
      JU    bLo2;
bEnd: NOP   0;
NETWORK
TITLE =  INIT_SECTION
      L     #CODE;
      L     3;
      <>I;
      JC    cEnd;
      S     DBX 45.7;	//"SecDB".ToASW.InfDataReady 
      S     DBX 44.1;	//"SecDB".ToASW.CmdNewBatch
      R     DBX 121.6;	//"SecDB".PCRead.Status.StaReset
      R     DBX 121.7;	//"SecDB".PCRead.Status.StaEndOfJob
      R     DBX 44.3;	//"SecDB".ToASW.InfSameJobPrevSec
      R     DBX 44.5;	//"SecDB".ToASW.InfSameBatchPrevSec
      R     DBX 44.4;	//"SecDB".ToASW.InfSameJobNextSec
      R     DBX 44.6;	//"SecDB".ToASW.InfSameBatchNextSec
      R     DBX 116.0;	//"SecDB".PCRead.Fault.EsBatchSize  [1C]
      L     0;
      T     DBD 202;	//"SecDB".JobAc.JobWeigth
      T     DBW 206;	//"SecDB".JobAc.BatchNo
      L     DBW 200;	//"SecDB".JobAc.StaBatch
      L     2#1000000000000000;
      AW;
      T     DBW 200;	//-->"SecDB".JobAc.StaBatch
      A     DBX 48.1;	// "SecDB".ToASW.Func.CmdAbortBatch
      S     DBX 201.0;	//->"SecDB".JobAc.StaBatch.StaErrBatch
      A     DBX 46.1;	// "SecDB".ToASW.Func.CmdEmptying
      S     DBX 200.6;	//--> "SecDB".JobAc.StaBatch.StaEmptyingBatch
      BEU;
cEnd: NOP   0;
NETWORK
TITLE =  Search section
//SUBROUTINE SEARCH SECTION:
//=======================
//INPUT : ACTUAL DB = Line-DB
//INPUT : LineDB.DBW20: SECTION-NR
//INPUT : LineDB DBW22: search_mode
//             0= Search section with equal section-Nr as DW10
//             1= Search first section with D22.15 ToASW.InfSameJobLineDB==1
//OUTPUT: LineDB DBW22: SECTION-DB
//        0== ILLEGAL SECTION-NR
      L     #CODE;
      L     4;
      <>I;
      JC    dEnd;
      OPN   DI [DBW 4];	//>>Call SecDB DI["LineDB".Para.ParFirstSecDB]
//LOOP:
dLop: L     DIW 2;	//"SecDB".Para.ParSecNr
      L     DBW 20;	//"LineDB".VarTemp[1]= Input.SectionNr.
      ==I;	//  
      AN    DBX 23.0;	//"LineDB".VarTemp[2]= Input.ModeFirstJob
      O;
      A     DBX 23.0;	//"LineDB".VarTemp[2]=Input.ModeFirstJob
      A     DIX 44.7;	//"SecDB".ToASW.InfSameJobLineDB
      JC    dOK;	//->found
      L     DIW 8;	//"SecDB".Para.ParNextSecDB
      L     0;
      ==I;
      JC    dErr;
      OPN   DI [DIW 8];	//--> Call next SecDB  DI["SecDB".Para.ParNextSecDB]
      JU    dLop;
//---End Loop ---
dOK:  L     DINO;	// Actual section DB
dErr: T     DBW 22;	//"LineDB".VarTemp[2] == output Section-DB (0=Not found)
      BEU;
dEnd: NOP   0;
NETWORK
TITLE =  search job
//SUBROUTINE SEARCH JOB:
//=======================
//SEARCH ALL SECTION WITH THE SAME JOB AS IN THE COMMUNICATION DB
//INPUT : ACTUAL DB = COM_DB
//OUTPUT: section-DB D22.15: ToASW.InfSameJobLineDB
//OUTPUT: "LineDB".DBX39.0 (VarTemp[10].0) = Job active
      L     #CODE;
      L     5;
      <>I;
      JC    eEnd;
      R     DBX 39.0;	//LineDB.VarTemp[10] : err_job_active      [1.4] 
      OPN   DI [DBW 4];	//>>Call 1.SecDB DI["LineDB".Para.ParFirstSecDB]
//LOOP:
eLop: SET;
      R     DIX 44.7;	//-->"SecDB".ToASW.InfSameJobLineDB
      A(;
      L     0;
      L     DBW 154;	//"LineDB".JobWrite.SectionDest
      ==I;
      O(;
      L     DIW 2;	//"SecDB".Para.ParSecNr
      ==I;
      );
      );
      A(;
      L     DID 160;	//"SecDB".JobNom.JobNr
      L     DBD 160;	//"LineDB".JobNom.JobNr
      ==D;
      A     DIX 45.7;	//"SecDB".ToASW.InfDataReady
      O(;
      A     DBX 145.0;	//"LineDB".JobWrite.Hsk.F_Define
      O     DBX 145.1;	// "LineDB".JobWrite.Hsk.F_Execute 
      AN    DIX 45.7;	//"SecDB".ToASW.InfDataReady
      );
      );
      =     DIX 44.7;	//-->"SecDB".ToASW.InfSameJobLineDB
      L     DID 160;	//"SecDB ".JobNom.JobNr                  [1.4]
      L     DBD 160;	//"LineDB".JobNom.JobNr                  [1.4]
      ==D;	//                                       [1.4]
      A     DIX 45.7;	//"SecDB".ToASW.InfDataReady             [1.4]
      S     DBX 39.0;	//-->LineDB.VarTemp[10]= err_job_active [1.4]
//Call next section
      L     DIW 8;	//SEC[i].Para.ParNextSecDB
      L     0;
      ==I;
      BEC;
      OPN   DI [DIW 8];	//DI["SecDB".Para.ParNextSecDBB]
      JU    eLop;
//---End Loop ---
eEnd: NOP   0;
NETWORK
TITLE =  CalcBatchSize (Code 6)
//SUBROUTINE TEST DONE:
//=======================
//SEARCH ALL SECTION WITH THE SAME JOB AS IN THE ACTAUL S_DB
//INPUT : ACTUAL DB = S_DB
//OUTPUT: D19.0: Job not found in a other section
//
//
      L     #CODE;
      L     6;
      <>I;
      JC    fEnd;
      L     DBW 168;	// "SecDB".JobNom.BatchNo
      T     DBW 208;	//->"SecDB".JobAc.BatchNoCal
      L     DBW 186;	// "SecDB".JobNom.BatchMaxPpm
      T     DBW 218;	// "SecDB".JobAc.BatchSizePpm
      L     DBW 168;	//  BatchNoTarget
      L     32767;	// 
      <>I;
      JC    fCAL;	// 
      L     DBD 164;	// "SecDB".JobNom.JobWeight
      L     DBD 202;	// "SecDB".JobAc.JobWeigth
      -D;	//  
      DTR;	// WtRest
      L     DBD 180;	// "SecDB".JobNom.BatchWeight
      DTR;	// 
      /R;	// 
      L     1.000000e+03;	// (promille)
      *R;	// 
      L     DBW 186;	// "SecDB".JobNom.BatchMaxPpm
      DTR;
      /R;
//      L     9.999990e-001
//      +R    
      RND+;	//  NrOfMaxBatch  [1D
      L     DBW 206;	//  "SecDB".JobAc.BatchNo
      +I;	// 
      T     DBW 208;	// ->"SecDB".JobAc.BatchNoCal
      L     DBD 164;	// "SecDB".JobNom.JobWeight
      L     DBD 202;	// "SecDB".JobAc.JobWeigth
      -D;	//  
      DTR;	// WtRest
      L     1.000000e+03;	// (promille)
      *R;	// 
      L     DBD 180;	// "SecDB".JobNom.BatchWeight==100%
      DTR;
      /R;
      RND;
      T     #VarRest;	// WtRest as  ppm
      L     DBW 184;	// "SecDB".JobNom.BatchMinPpm
      <=D;
      A     DBX 201.3;	// "SecDB".JobAc.StaBatch.StaLastBatch
      JC    fDON;	//  -> job done
      <D;	// [Rel 1.5]
      L     #VarRest;	// WtRest as ppm
      JC    fERO;	// ->Fault: EsBatchSize
// Test 1 batches left 
      L     DBW 186;	// "SecDB".JobNom.BatchMaxPpm
      <=D;
      JC    fRST;	// --> Rest
// Test 2 batches left 
      SLD   1;	// 2* batchMaxPc
      <=D;	// 
      JC    fHAF;	// -> batch:= Rest/2
// Maximum Batch
      L     #VarRest;	// WtRestPc as ppm
      L     DBW 186;	// "SecDB".JobNom.BatchMaxPpm
      -D;	// 
      L     DBW 184;	// "SecDB".JobNom.BatchMinPpm
      SLD   1;	// 2*batchMinPc
      >=D;	// 
      L     DBW 186;	// "SecDB".JobNom.BatchMaxPpm
      JC    fSIZ;	// -> batch := "SecDB".JobNom.BatchMaxPpm
// Test 3 batches left
      L     DBW 206;	// "SecDB".JobAc.BatchNo
      +     3;	// 
      T     DBW 208;	// ->"SecDB".JobAc.BatchNoCal
      L     #VarRest;	// 
      DTR;	// 
      L     3.000000e+00;	//   /3
      /R;	// 
      RND;	// VarBatchSizePc
      L     DBW 184;	//  "SecDB".JobNom.BatchMinPpm
      <I;	// 
      JC    fSIZ;	//->Start minimum Size
      TAK;	// 
      JU    fSIZ;	//->Batch Size = Rest/3
fHAF: L     #VarRest;
      SSD   1;	//  /2
      L     DBW 184;	//  "SecDB".JobNom.BatchMinPpm
      >=I;
      TAK;
      JC    fSIZ;	// -> Batch Size = Rest/2
      JU    fERO;
//== Error =====================
fERO: T     DBW 218;	//"SecDB".JobAc.BatchSizePpm
      A     DBX 47.7;	// "SecDB".ToASW.Func.CmdAcceptSize
      JC    fSIZ;	// 
      AN    DBX 116.0;	// "SecDB".PCRead.Fault.EsBatchSize
      S     DBX 116.0;	// -> "SecDB".PCRead.Fault.EsBatchSize
      S     DBX 48.3;	// ->"SecDB".ToASW.Func.CmdHornOn
      JU    fCAL;
// === Start Batch ===============
//Error batch size
fDON: R     DBX 116.0;	// -> "SecDB".PCRead.Fault.EsBatchSize  
      S     DBX 121.7;	// ->"SecDB".PCRead.Status.StaEndOfJob
      L     DBW 206;	//  "SecDB".JobAc.BatchNo 
      T     DBW 208;	// ->"SecDB".JobAc.BatchNoCal
      BEU;
//Last Batch
fRST: S     DBX 201.3;	//->"SecDB".JobAc.StaBatch.StaLastBatch
      L     #VarRest;	//var_WtRestPc
fSIZ: T     DBW 218;	//-->"SecDB".JobAc.BatchSizePpm
      R     DBX 116.0;	//-> "SecDB".PCRead.Fault.EsBatchSize
fCAL: L     DBW 218;	//"SecDB".JobAc.BatchSizePpm
      DTR;	// 
      L     DBD 180;	// "SecDB".JobNom.BatchWeight
      DTR;	// 
      *R;	// 
      L     1.000000e+03;	// [1/1000]
      /R;	// 
      RND;	// 
      T     DBD 210;	// ->"SecDB".JobAc.BatchWeigthTarget
      BEU;
fEnd: NOP   0;
NETWORK
TITLE =  TestDone Code 7)
      L     #CODE;	// 
      L     7;	// 
      <>I;	// 
      JC    gEnd;	// 
      S     DBX 39.0;	// outp_NotFound
      OPN   DI [DBW 4];	//>>call LineDB  DI["SecDB".Para.ParLineDB]
      OPN   DI [DIW 4];	//>>Call 1.SecDB DI["LineDB".Para.ParFirstSecDB]
//Loop over all section
gLop: L     DID 160;	// SecDB[i].JobNom.JobNr
      L     DBD 160;	// "SecDB".JobNom.JobNr
      <>D;	// 
      ON    DIX 45.7;	// "SecDB".ToASW.InfDataReady
      JC    gNeq;	// 
      L     DINO;	// SecDB[i]
      L     DBNO;	// SecDB
      <>I;	// 
      R     DBX 39.0;	// outp_NotFound
gNeq: L     DIW 8;	// SecDB[i].Para.ParNextSecDB
      L     0;	// 
      ==I;	// 
      BEC;	// 
//-->Call next SecDB  DI["SecDB".Para.ParNextSecDB]
      OPN   DI [DIW 8];
      JU    gLop;
//---End Loop ---
gEnd: NOP   0;
NETWORK
TITLE =
END_FUNCTION

FUNCTION "Takt/Pause" : VOID	// FC 1105
VERSION : 0.1
VAR_INPUT
  ProzesszeitMin : INT ;
  StartMin : INT ;
  Dauer : INT ;
  Anzahl_Takt : INT ;
  Teiler_Pause : INT ;
  Typ_TaktPause : BOOL ;
END_VAR
VAR_OUTPUT
  Run1 : BOOL ;
  Run2 : BOOL ;
  Run3 : BOOL ;
  Run4 : BOOL ;
  Run5 : BOOL ;
  Run6 : BOOL ;
END_VAR
VAR_TEMP
  TimeInActPeriod : INT ;
  TimeInActPeriod1ST : INT ;
  DurationActPeriod : INT ;
  TimeInIntervall : INT ;
  OnTimeInIntervall : INT ;
END_VAR
BEGIN
NETWORK
TITLE =
// (network holds code this reader does not know; not shown)
//      L     #Dauer
//      L     #DurationActPeriod
//      MOD   
// Laufsignal Nr1
// Laufsignal Nr2
// Laufsignal Nr3
// Laufsignal Nr4
// Laufsignal Nr5
// Laufsignal Nr6
//      Takt_Pause
// Laufsignal Nr1
END_FUNCTION

FUNCTION "Takt mit Pause" : VOID	// FC 1106
VERSION : 0.1
VAR_INPUT
  ProzesszeitMin : INT ;
  StartMin : INT ;
  Dauer : INT ;
  Anzahl_Takt : INT ;
  Teiler_Pause : INT ;
  Typ_TaktPause : BOOL ;
END_VAR
VAR_OUTPUT
  Run1 : BOOL ;
  Run2 : BOOL ;
  Run3 : BOOL ;
  Run4 : BOOL ;
  Run5 : BOOL ;
  Run6 : BOOL ;
END_VAR
VAR_TEMP
  TimeInActPeriod : INT ;
  TimeInActPeriod1ST : INT ;
  DurationActPeriod : INT ;
  TimeInIntervall : INT ;
  OnTimeInIntervall : INT ;
END_VAR
BEGIN
NETWORK
TITLE =
// (network holds code this reader does not know; not shown)
//      L     #Dauer
// Laufsignal Nr1
// Laufsignal Nr2
// Laufsignal Nr3
// Laufsignal Nr4
// Laufsignal Nr5
// Laufsignal Nr6
//- Takt_Pause ---
// Laufsignal Nr1
END_FUNCTION

DATA_BLOCK "EventsToPIC_DB"	// DB 470
VERSION : 0.0
"SSA_MH_EventsToPIC"
BEGIN
END_DATA_BLOCK

DATA_BLOCK "SSA_LOG_Value_Queue"	// DB 1005
TITLE = SYS_LOG_Queue
//COPYRIGHT:    (C) 1996 BY  BUHLER LTD.
//                           CH-9240 UZWIL  SWITZERLAND
//
//PRODUCT:      GCS90_OS.LOG
//
//TITLE:        QUEUE-DB
//
//-------------------------------------------------------------------------
//
//IDENT:        AUTOR:              DEPT:                       DATE:
//
//DB5.1A        S. Kalberer         AEE61                       4-Jun-1996
//              1st Release in S7, converted from DB220.1A
//
//-------------------------------------------------------------------------
//
//PURPOSE:      MANUAL : LOGMAN
//              CODE   : FB46,47
//
//RESTRICTIONS: S7
//              only for PC-Interface
//
//-------------------------------------------------------------------------
//
//
AUTHOR : SK
FAMILY : GCS7SYS
NAME : LOG_DB
VERSION : 0.0
  STRUCT
   Fault : WORD ;	//Bit 0 Fault Block copy
   ParByteReadQueuePC : INT  := 60;	//1st Byte to Read the Queue from the PC
   ParByteLenghtMessage : INT  := 200;	//Lenght of Message Block in Queue
   ParMaxNoOfMsg : INT  := 200;	//Max index of array MsgQueue
   VarNrOfMsgInQueue : INT ;	//Actual number of Msg in queue
   VarByteWrite : WORD ;	//Write pointer
   VarByteRead : WORD ;	//Read pointer
   ParByteLenghtUDT : INT  := 200;	//1st Byte or ParMsgFull
   ParStartFIFO : INT  := 660;	//First Byte of the Queue
   ParStartMessageFull : INT  := 260;
   ParStartInput : INT  := 460;	//Used for ASW to send an inputmessage to Queue
   Spare22 : INT ;
   Spare24 : INT ;
   Spare26 : INT ;
   Spare28 : INT ;
   Spare30 : INT ;
   Spare32 : INT ;
   Spare34 : INT ;
   Spare36 : INT ;
   Spare38 : INT ;
   ChangeBit : STRUCT
    spare : BYTE ;
    CBit0 : BOOL ;
   END_STRUCT ;
   ParNrOfMsgMemory : INT  := 1;	//Max index of array PC.Msg
   spare : BYTE ;
   ParPC1Connected : BOOL  := TRUE;	//Pc1 is connected
   ParPC2Connected : BOOL ;	//Pc1 is connected
   ParPC3Connected : BOOL ;	//Pc1 is connected
   ParPC4Connected : BOOL ;	//Pc1 is connected
   spare4504 : BOOL ;
   spare4505 : BOOL ;
   spare4506 : BOOL ;
   spare4507 : BOOL ;
   spare4600 : BOOL ;
   spare4601 : BOOL ;
   spare4602 : BOOL ;
   spare4603 : BOOL ;
   spare4604 : BOOL ;
   spare4605 : BOOL ;
   CmdAddFastMsg : BOOL ;	//->Add Fast Message directly at PC interface
   CmdResetLog : BOOL  := TRUE;	//->Init Queue
   InPC1Online : BOOL ;	//->PC1 is offline
   InPC2Online : BOOL ;	//->PC2 is offline
   InPC3Online : BOOL ;	//->PC3 is offline
   InPC4Online : BOOL ;	//->PC4 is offline
   PC : STRUCT 	//=== Interface to PC
    HskPC1toPLC : WORD ;
    HskPC2toPLC : WORD ;
    HskPC3toPLC : WORD ;
    HskPC4toPLC : WORD ;
    HskPLCtoPC : WORD ;
    NrOfMessageInQueue : WORD  := W#16#1;
    Read : ARRAY  [1 .. 1 ] OF //Message for PC
    STRUCT
     Message : UDT 10005;
    END_STRUCT ;
   END_STRUCT ;
   ParMsgFull : UDT 10005;	//===Message queue full
   Input : UDT 10005;	//===Input to Message queue
   MsgQueue : ARRAY  [1 .. 200 ] OF UDT 10005;
  END_STRUCT ;	
BEGIN
   ParByteReadQueuePC := 60;
   ParByteLenghtMessage := 200;
   ParMaxNoOfMsg := 200;
   ParByteLenghtUDT := 200;
   ParStartFIFO := 660;
   ParStartMessageFull := 260;
   ParStartInput := 460;
   ParNrOfMsgMemory := 1;
   ParPC1Connected := TRUE;
   CmdResetLog := TRUE;
   PC.NrOfMessageInQueue := W#16#1;
END_DATA_BLOCK

DATA_BLOCK "DB Prozesszeit"	// DB 1010
VERSION : 0.1
  STRUCT
   DB_VAR : INT ;	//vorläufige Platzhaltervariable
   ErsteSektion : INT  := 1;	//Startwert, bei welcher Sektion begonnen wird
   Anzahl_Sektionen : INT  := 16;	//16 Sektionen, kann bei Bedarf verringert werden, Startwert beachten
   Zaehler : INT  := 1;	//Zähler Sektionsnummer
   ZeigerLesenSchreiben : INT  := 70;	//Start 1. Sektion
   Arbeitsbereich : STRUCT
    dt1 : DATE_AND_TIME ;	//Startzeit
    dt2 : DATE_AND_TIME ;	//Aktuelle Zeit
    dt12 : DATE_AND_TIME ;
    Diff : TIME ;	//aktuelle Prozesszeit
    temp1 : INT ;
    Prozess_aktiv : BOOL ;
    Bit01 : BOOL ;
    Bit02 : BOOL ;
    Bit03 : BOOL ;
    Bit04 : BOOL ;
    Bit05 : BOOL ;
    Bit06 : BOOL ;
    Bit07 : BOOL ;
    Byte0 : BYTE ;
    Tage : INT ;
    Stunden : INT ;
    Minuten : INT ;
    Rest : DINT ;
    Sekunden : INT ;
    Pointer_10min : INT ;
    Pointer_30min : INT ;
    Pointer_90min : INT ;
    Visu_Tage : INT ;
    Visu_StundenProTag : INT ;
    Visu_MinutenProStunde : INT ;
    Gesamtzeit_in_Minuten : INT ;
    Res_int01 : INT ;
   END_STRUCT ;
   Sektion_1 : STRUCT
    dt1 : DATE_AND_TIME ;
    dt2 : DATE_AND_TIME ;
    dt12 : DATE_AND_TIME ;
    Diff : TIME ;
    temp1 : INT ;
    Prozess_aktiv : BOOL ;
    Bit01 : BOOL ;
    Bit02 : BOOL ;
    Bit03 : BOOL ;
    Bit04 : BOOL ;
    Bit05 : BOOL ;
    Bit06 : BOOL ;
    Bit07 : BOOL ;
    Byte0 : BYTE ;
    Tage : INT ;
    Stunden : INT ;
    Minuten : INT ;
    Rest : DINT ;
    Sekunden : INT ;
    Pointer_10min : INT ;
    Pointer_30min : INT ;
    Pointer_90min : INT ;
    Visu_Tage : INT ;
    Visu_StundenProTag : INT ;
    Visu_MinutenProStunde : INT ;
    Gesamtzeit_in_Minuten : INT ;
    Res_int01 : INT ;
   END_STRUCT ;
   Sektion_3 : STRUCT
    dt1 : DATE_AND_TIME ;
    dt2 : DATE_AND_TIME ;
    dt12 : DATE_AND_TIME ;
    Diff : TIME ;
    temp1 : INT ;
    Prozess_aktiv : BOOL ;
    Bit01 : BOOL ;
    Bit02 : BOOL ;
    Bit03 : BOOL ;
    Bit04 : BOOL ;
    Bit05 : BOOL ;
    Bit06 : BOOL ;
    Bit07 : BOOL ;
    Byte0 : BYTE ;
    Tage : INT ;
    Stunden : INT ;
    Minuten : INT ;
    Rest : DINT ;
    Sekunden : INT ;
    Pointer_10min : INT ;
    Pointer_30min : INT ;
    Pointer_90min : INT ;
    Visu_Tage : INT ;
    Visu_StundenProTag : INT ;
    Visu_MinutenProStunde : INT ;
    Gesamtzeit_in_Minuten : INT ;
    Res_int01 : INT ;
   END_STRUCT ;
   Sektion_5 : STRUCT
    dt1 : DATE_AND_TIME ;
    dt2 : DATE_AND_TIME ;
    dt12 : DATE_AND_TIME ;
    Diff : TIME ;
    temp1 : INT ;
    Prozess_aktiv : BOOL ;
    Bit01 : BOOL ;
    Bit02 : BOOL ;
    Bit03 : BOOL ;
    Bit04 : BOOL ;
    Bit05 : BOOL ;
    Bit06 : BOOL ;
    Bit07 : BOOL ;
    Byte0 : BYTE ;
    Tage : INT ;
    Stunden : INT ;
    Minuten : INT ;
    Rest : DINT ;
    Sekunden : INT ;
    Pointer_10min : INT ;
    Pointer_30min : INT ;
    Pointer_90min : INT ;
    Visu_Tage : INT ;
    Visu_StundenProTag : INT ;
    Visu_MinutenProStunde : INT ;
    Gesamtzeit_in_Minuten : INT ;
    Res_int01 : INT ;
   END_STRUCT ;
   Sektion_6 : STRUCT
    dt1 : DATE_AND_TIME ;
    dt2 : DATE_AND_TIME ;
    dt12 : DATE_AND_TIME ;
    Diff : TIME ;
    temp1 : INT ;
    Prozess_aktiv : BOOL ;
    Bit01 : BOOL ;
    Bit02 : BOOL ;
    Bit03 : BOOL ;
    Bit04 : BOOL ;
    Bit05 : BOOL ;
    Bit06 : BOOL ;
    Bit07 : BOOL ;
    Byte0 : BYTE ;
    Tage : INT ;
    Stunden : INT ;
    Minuten : INT ;
    Rest : DINT ;
    Sekunden : INT ;
    Pointer_10min : INT ;
    Pointer_30min : INT ;
    Pointer_90min : INT ;
    Visu_Tage : INT ;
    Visu_StundenProTag : INT ;
    Visu_MinutenProStunde : INT ;
    Gesamtzeit_in_Minuten : INT ;
    Res_int01 : INT ;
   END_STRUCT ;
   Sektion_7 : STRUCT
    dt1 : DATE_AND_TIME ;
    dt2 : DATE_AND_TIME ;
    dt12 : DATE_AND_TIME ;
    Diff : TIME ;
    temp1 : INT ;
    Prozess_aktiv : BOOL ;
    Bit01 : BOOL ;
    Bit02 : BOOL ;
    Bit03 : BOOL ;
    Bit04 : BOOL ;
    Bit05 : BOOL ;
    Bit06 : BOOL ;
    Bit07 : BOOL ;
    Byte0 : BYTE ;
    Tage : INT ;
    Stunden : INT ;
    Minuten : INT ;
    Rest : DINT ;
    Sekunden : INT ;
    Pointer_10min : INT ;
    Pointer_30min : INT ;
    Pointer_90min : INT ;
    Visu_Tage : INT ;
    Visu_StundenProTag : INT ;
    Visu_MinutenProStunde : INT ;
    Gesamtzeit_in_Minuten : INT ;
    Res_int01 : INT ;
   END_STRUCT ;
   Sektion_8 : STRUCT
    dt1 : DATE_AND_TIME ;
    dt2 : DATE_AND_TIME ;
    dt12 : DATE_AND_TIME ;
    Diff : TIME ;
    temp1 : INT ;
    Prozess_aktiv : BOOL ;
    Bit01 : BOOL ;
    Bit02 : BOOL ;
    Bit03 : BOOL ;
    Bit04 : BOOL ;
    Bit05 : BOOL ;
    Bit06 : BOOL ;
    Bit07 : BOOL ;
    Byte0 : BYTE ;
    Tage : INT ;
    Stunden : INT ;
    Minuten : INT ;
    Rest : DINT ;
    Sekunden : INT ;
    Pointer_10min : INT ;
    Pointer_30min : INT ;
    Pointer_90min : INT ;
    Visu_Tage : INT ;
    Visu_StundenProTag : INT ;
    Visu_MinutenProStunde : INT ;
    Gesamtzeit_in_Minuten : INT ;
    Res_int01 : INT ;
   END_STRUCT ;
   Sektion_17 : STRUCT
    dt1 : DATE_AND_TIME ;
    dt2 : DATE_AND_TIME ;
    dt12 : DATE_AND_TIME ;
    Diff : TIME ;
    temp1 : INT ;
    Prozess_aktiv : BOOL ;
    Bit01 : BOOL ;
    Bit02 : BOOL ;
    Bit03 : BOOL ;
    Bit04 : BOOL ;
    Bit05 : BOOL ;
    Bit06 : BOOL ;
    Bit07 : BOOL ;
    Byte0 : BYTE ;
    Tage : INT ;
    Stunden : INT ;
    Minuten : INT ;
    Rest : DINT ;
    Sekunden : INT ;
    Pointer_10min : INT ;
    Pointer_30min : INT ;
    Pointer_90min : INT ;
    Visu_Tage : INT ;
    Visu_StundenProTag : INT ;
    Visu_MinutenProStunde : INT ;
    Gesamtzeit_in_Minuten : INT ;
    Res_int01 : INT ;
   END_STRUCT ;
   Sektion_33 : STRUCT
    dt1 : DATE_AND_TIME ;
    dt2 : DATE_AND_TIME ;
    dt12 : DATE_AND_TIME ;
    Diff : TIME ;
    temp1 : INT ;
    Prozess_aktiv : BOOL ;
    Bit01 : BOOL ;
    Bit02 : BOOL ;
    Bit03 : BOOL ;
    Bit04 : BOOL ;
    Bit05 : BOOL ;
    Bit06 : BOOL ;
    Bit07 : BOOL ;
    Byte0 : BYTE ;
    Tage : INT ;
    Stunden : INT ;
    Minuten : INT ;
    Rest : DINT ;
    Sekunden : INT ;
    Pointer_10min : INT ;
    Pointer_30min : INT ;
    Pointer_90min : INT ;
    Visu_Tage : INT ;
    Visu_StundenProTag : INT ;
    Visu_MinutenProStunde : INT ;
    Gesamtzeit_in_Minuten : INT ;
    Res_int01 : INT ;
   END_STRUCT ;
   Sektion_34 : STRUCT
    dt1 : DATE_AND_TIME ;
    dt2 : DATE_AND_TIME ;
    dt12 : DATE_AND_TIME ;
    Diff : TIME ;
    temp1 : INT ;
    Prozess_aktiv : BOOL ;
    Bit01 : BOOL ;
    Bit02 : BOOL ;
    Bit03 : BOOL ;
    Bit04 : BOOL ;
    Bit05 : BOOL ;
    Bit06 : BOOL ;
    Bit07 : BOOL ;
    Byte0 : BYTE ;
    Tage : INT ;
    Stunden : INT ;
    Minuten : INT ;
    Rest : DINT ;
    Sekunden : INT ;
    Pointer_10min : INT ;
    Pointer_30min : INT ;
    Pointer_90min : INT ;
    Visu_Tage : INT ;
    Visu_StundenProTag : INT ;
    Visu_MinutenProStunde : INT ;
    Gesamtzeit_in_Minuten : INT ;
    Res_int01 : INT ;
   END_STRUCT ;
  END_STRUCT ;	
BEGIN
   ErsteSektion := 1;
   Anzahl_Sektionen := 16;
   Zaehler := 1;
   ZeigerLesenSchreiben := 70;
END_DATA_BLOCK

SYMBOL_TABLE
"PLC_SystemDB"	DB 50	DB 50	// PLC: System informations
"PC_StorageDB"	DB 53	DB 53	// PC: Storage with free assignment
"ASW_TimerSettings"	DB 56	DB 56	// USW: Timer settings
"ASW_GraphicData"	DB 80	DB 80
"ASW_PlantParData"	DB 81	DB 81
"ASW_LineInfoData"	DB 82	DB 82
"ASW_HandAddInfoData"	DB 83	DB 83
"PCC_YieldScaleDB"	DB 90	DB 90	// PCC: Databuffer for PCC yield calculation
"ASW_DFCATargData"	DB 480	DB 480
"PLC1Snd"	DB 1711	DB 1711	// COM: Send data to PLC 1
"PLC2Snd"	DB 1712	DB 1712	// COM: Send data to PLC 2
"PLC3Snd"	DB 1713	DB 1713	// COM: Send data to PLC 3
"PLC4Snd"	DB 1714	DB 1714	// COM: Send data to PLC 4
"PLC5Snd"	DB 1715	DB 1715	// COM: Send data to PLC 5
"PLC1Rcv"	DB 1721	DB 1721	// COM: Receive data from PLC 1
"PLC2Rcv"	DB 1722	DB 1722	// COM: Receive data from PLC 2
"PLC3Rcv"	DB 1723	DB 1723	// COM: Receive data from PLC 3
"PLC4Rcv"	DB 1724	DB 1724	// COM: Receive data from PLC 4
"PLC5Rcv"	DB 1725	DB 1725	// COM: Receive data from PLC 5
"ComPLC1Snd"	DB 1761	FB 1701	// COM: Send buffer PLC 1
"ComPLC2Snd"	DB 1762	FB 1701	// COM: Send buffer PLC 2
"ComPLC3Snd"	DB 1763	FB 1701	// COM: Send buffer PLC 3
"ComPLC4Snd"	DB 1764	FB 1701	// COM: Send buffer PLC 4
"ComPLC5Snd"	DB 1765	FB 1701	// COM: Send buffer PLC 5
"ComPLC1Rcv"	DB 1771	FB 1702	// COM: Receive buffer PLC 1
"ComPLC2Rcv"	DB 1772	FB 1702	// COM: Receive buffer PLC 2
"ComPLC3Rcv"	DB 1773	FB 1702	// COM: Receive buffer PLC 3
"ComPLC4Rcv"	DB 1774	FB 1702	// COM: Receive buffer PLC 4
"ComPLC5Rcv"	DB 1775	FB 1702	// COM: Receive buffer PLC 5
"T_FMODEMON"	DB 4001	DB 4001	// Only for TEST reasons.
"STD_LineSecStdSub2"	FB 90	FB 90	// STD: Line and section control standard subroutines
"TON_BREAK"	FB 1704	FB 1704	// IEC-TON timer with break functionality
"T_BREAK"	FB 1706	FB 1706	// IEC-TOF timer with break functionality
"STD_PULSEGEN"	FB 1707	FB 1707	// Buhler pulse generator
"STD_BranIntermitted"	FB 1802	FB 1802	// STD: Intermitted mode of bransilos
"STD_DryIntervalFilling"	FB 1803	FB 1803	// STD: Dry- and interval filling for wheat bins
"STD_DUMPFlowMonitor"	FB 1804	FB 1804	// STD: DUMP-Scale test productflow
"STD_DUMPPulse"	FB 1805	FB 1805	// STD: Handling of Scales with Dump Impuls
"D_TOD_DT"	FC 3	FC 3	// Date and TOD to DT
"DT_DATE"	FC 6	FC 6	// DT to DATE
"DT_TOD"	FC 8	FC 8	// DT to TOD
"SYS_CallLineSection"	FC 11	FC 11	// SYS: Call line and section controller
"LOG_GCS90_convert"	FC 45	FC 45	// LOG: GCS90 message convert
"LOG_EntryQueue"	FC 46	FC 46	// LOG: Message entry in queue
"SYS_DPDiag1"	FC 76	FC 76	// DPDiagnose => not Siemens Slave
"ASW_GraphicFunction"	FC 80	FC 80
"ASW_PlantParFunction"	FC 81	FC 81
"SIEMENS.IECFC6.DT_DATE"	FC 90	FC 90
"SIEMENSTOD_DT"	FC 91	FC 91
"SIEMENS.IECFC3.TOD_DT"	FC 92	FC 92
"SIEMENS.IECFC10.EQ_STR"	FC 93	FC 93
"SYS_GeneralPLCStartup"	FC 100	FC 100	// SYS: General plc startup functions
"SYS_GeneralFunctions"	FC 105	FC 105	// SYS: General plant signals
"TEST_Functions"	FC 111	FC 111	// TEST: Testfunctions
"STD_LineSecStdSub"	FC 120	FC 120	// STD: Line and section control standard subroutines
"STD_OnOffSignals32"	FC 122	FC 122	// STD: ON / OFF Signal handling with 32-Bit
"COM_PLCtoPLC"	FC 141	FC 141	// COM: PLC to PLC communication
"STD_SearchChangeBit"	FC 241	FC 241	// STD: Search object change bits
"STD_PLCLiveValue"	FC 242	FC 242	// STD: Live value handling for PCC
"STD_AuxiliaryFunctions"	FC 247	FC 247	// STD: Auxiliary functions
"STD_EdgeFunctions"	FC 248	FC 248	// STD: Edge / step functions
"STD_ScaleAnalogSignal"	FC 249	FC 249	// STD: Convert SIEMENS S5 analog values
"CPU_CopyPulse100ms"	M 1.0	BOOL	// CPU: System timing
"CPU_CopyPulse200ms"	M 1.1	BOOL	// CPU: System timing
"CPU_CopyPulse400ms"	M 1.2	BOOL	// CPU: System timing
"CPU_CopyPulse500ms"	M 1.3	BOOL	// CPU: System timing
"CPU_CopyPulse800ms"	M 1.4	BOOL	// CPU: System timing
"CPU_CopyPulse1000ms"	M 1.5	BOOL	// CPU: System timing
"CPU_CopyPulse1600ms"	M 1.6	BOOL	// CPU: System timing
"CPU_CopyPulse1800ms"	M 1.7	BOOL	// CPU: System timing
"CPU_Pulse100ms"	M 2.0	BOOL	// CPU: System timing
"CPU_Pulse200ms"	M 2.1	BOOL	// CPU: System timing
"CPU_Pulse400ms"	M 2.2	BOOL	// CPU: System timing
"CPU_Pulse500ms"	M 2.3	BOOL	// CPU: System timing
"CPU_Pulse800ms"	M 2.4	BOOL	// CPU: System timing
"CPU_Pulse1000ms"	M 2.5	BOOL	// CPU: System timing
"CPU_Pulse1600ms"	M 2.6	BOOL	// CPU: System timing
"CPU_Pulse2000ms"	M 2.7	BOOL	// CPU: System timing
"SYS_ScanA_IsOn"	M 3.1	BOOL	// SYS: Scan A is active
"SYS_ScanB_IsOn"	M 3.2	BOOL	// SYS: Scan B is active
"SYS_ScanC_IsOn"	M 3.3	BOOL	// SYS: Scan C is active
"SYS_Scan0_Tick100ms"	M 4.2	BOOL	// SYS_Scan0: Is every 100ms for one scan high
"SYS_Scan0_Tick200ms"	M 4.3	BOOL	// SYS_Scan0: Is every 200ms for one scan high
"SYS_Scan0_Tick500ms"	M 4.4	BOOL	// SYS_Scan0: Is every 500ms for one scan high
"SYS_Scan0_Tick1s"	M 4.5	BOOL	// SYS_Scan0: Is every 1s for one scan high
"SYS_Scan0_Tick1min"	M 4.6	BOOL	// SYS_Scan0: Is every min for one scan high
"SYS_ScanA_Tick200ms"	M 5.3	BOOL	// SYS_ScanA: Is every 200ms for one scan high
"SYS_ScanA_Tick500ms"	M 5.4	BOOL	// SYS_ScanA:  Is every 500ms for one scan high
"SYS_ScanA_Tick1s"	M 5.5	BOOL	// SYS_ScanA: Is every 1s for one scan high
"SYS_ScanA_Tick1min"	M 5.6	BOOL	// SYS_ScanA: Is every min for one scan high
"SYS_ScanB_Tick200ms"	M 6.3	BOOL	// SYS_ScanB: Is every 200ms for one scan high
"SYS_ScanB_Tick500ms"	M 6.4	BOOL	// SYS_ScanB: Is every 500ms for one scan high
"SYS_ScanB_Tick1s"	M 6.5	BOOL	// SYS_ScanB: Is every 1s for one scan high
"SYS_ScanB_Tick1min"	M 6.6	BOOL	// SYS_ScanB: Is every min for one scan high
"SYS_ScanC_Tick200ms"	M 7.3	BOOL	// SYS_ScanC: Is every 200ms for one scan high
"SYS_ScanC_Tick500ms"	M 7.4	BOOL	// SYS_ScanC: Is every 500ms for one scan high
"SYS_ScanC_Tick1s"	M 7.5	BOOL	// SYS_ScanC: Is every 1s for one scan high
"SYS_ScanC_Tick1min"	M 7.6	BOOL	// SYS_ScanC: Is every min for one scan high
"SYS_infLog0"	M 9.0	BOOL	// SYS: Logical false all the time
"SYS_infLog1"	M 9.1	BOOL	// SYS: Logical true all the time
"SYS_CycleFlasher"	M 9.2	BOOL	// SYS: Status changing every scan
"SYS_Pulse500ms"	M 9.3	BOOL	// SYS: Pulse 500 ms true, 500ms false
"SYS_Pulse1000ms"	M 9.4	BOOL	// SYS: Pulse 1000ms true, 1000ms false
"SYS_Tick1s"	M 9.5	BOOL	// SYS: Tick is every 1s for one scan high
"SYS_MainProgram"	OB 1	OB 1	// SYS: Main program
"SYS_CycInt20ms"	OB 35	OB 35	// SYS: Cyclic interrupt 20 ms
"SYS_PS_FLT"	OB 81	OB 81	// SYS: Power Supply Fault
"SYS_IO_FLT"	OB 82	OB 82	// SYS: I/O Point Fault
"SYS_RACK_FLT"	OB 86	OB 86	// SYS: Loss of Rack Fault
"PLC_StUpNewstart"	OB 100	OB 100	// PLC: Startup program on newstart
"PLC_StUpRestart"	OB 101	OB 101	// PLC: Startup program on restart
"PLC_StUpColdstart"	OB 102	OB 102	// PLC: Startup program on coldstart
"SYS_MOD_ERR"	OB 122	OB 122	// SYS: Module Access Error
"CTUD"	SFB 2	SFB 2	// Count Up / Down
"BSEND"	SFB 12	SFB 12	// Sending Segmented Data
"BRCV"	SFB 13	SFB 13	// Receiving Segmented Data
"REPL_VAL"	SFC 44	SFC 44	// Transfer Substitute Value to Accumulator 1
"T_ResetHeavyStartupFlag"	T 16	TIMER	// SYS: Reset the "GCS7_Gr_InHeavyStartup" (M13.6) after this time
"ASW_Flags_F0_F15"	UDT 1000	UDT 1000
"ASW_LineAnimation"	UDT 1001	UDT 1001
"ASW_UserSectionState"	UDT 1002	UDT 1002
"ASW_ProductInfo"	UDT 1003	UDT 1003
"ASW_HandAddInfo"	UDT 1004	UDT 1004
"ASW_DFCARecipe"	UDT 1005	UDT 1005
"STD_BinProteinControl"	UDT 1201	UDT 1201	// STD: Bin status protein controller
"GCS7_UDT_FunctionKey"	UDT 10601	UDT 10601	// GCS7: Upper Layer
"GCS7_UDT_FaultPattern"	UDT 10602	UDT 10602	// GCS7: Upper Layer
"GCS7_UDT_StatusPattern"	UDT 10603	UDT 10603	// Upper Layer
"MELEYieldScale"	UDT 19000	UDT 19000	// USW: Struct for scales involved in yield calculation
"WinCoSYieldScale"	UDT 19001	UDT 19001	// USW: Struct for scales involved in yield calculation
"SamplerData"	UDT 19002	UDT 19002	// USW: Struct for samplers
"BigBagData"	UDT 19003	UDT 19003	// Registration of big bag weight
"GCS7_FB9_Communication"	UDT 20099	UDT 20099	// Communication PLC --PLC
"VAT_GCS7System"	VAT 1		// VAT: System flags from GCS90
"VAT_System"	VAT 2		// VAT: System flags from user software
"VAT_PLCCommunication"	VAT 3		// VAT: PLC to PLC communication overview
"VAT_Diagnosis"	VAT 4		// VAT: PLC diagnosis
END_SYMBOL_TABLE

TYPE "ASW_Flags_F0_F15"	// UDT 1000
VERSION : 0.0
  STRUCT
   F8 : BOOL ;
   F9 : BOOL ;
   F10 : BOOL ;
   F11 : BOOL ;
   F12 : BOOL ;
   F13 : BOOL ;
   F14 : BOOL ;
   F15 : BOOL ;
   F0 : BOOL ;
   F1 : BOOL ;
   F2 : BOOL ;
   F3 : BOOL ;
   F4 : BOOL ;
   F5 : BOOL ;
   F6 : BOOL ;
   F7 : BOOL ;
  END_STRUCT ;	
END_TYPE

TYPE "ASW_LineAnimation"	// UDT 1001
VERSION : 0.0
  STRUCT
   L0 : STRUCT
    B8 : BOOL ;
    B9 : BOOL ;
    B10 : BOOL ;
    B11 : BOOL ;
    B12 : BOOL ;
    B13 : BOOL ;
    B14 : BOOL ;
    B15 : BOOL ;
    B0 : BOOL ;
    B1 : BOOL ;
    B2 : BOOL ;
    B3 : BOOL ;
    B4 : BOOL ;
    B5 : BOOL ;
    B6 : BOOL ;
    B7 : BOOL ;
   END_STRUCT ;
   L1 : STRUCT
    B8 : BOOL ;
    B9 : BOOL ;
    B10 : BOOL ;
    B11 : BOOL ;
    B12 : BOOL ;
    B13 : BOOL ;
    B14 : BOOL ;
    B15 : BOOL ;
    B0 : BOOL ;
    B1 : BOOL ;
    B2 : BOOL ;
    B3 : BOOL ;
    B4 : BOOL ;
    B5 : BOOL ;
    B6 : BOOL ;
    B7 : BOOL ;
   END_STRUCT ;
   L2 : STRUCT
    B8 : BOOL ;
    B9 : BOOL ;
    B10 : BOOL ;
    B11 : BOOL ;
    B12 : BOOL ;
    B13 : BOOL ;
    B14 : BOOL ;
    B15 : BOOL ;
    B0 : BOOL ;
    B1 : BOOL ;
    B2 : BOOL ;
    B3 : BOOL ;
    B4 : BOOL ;
    B5 : BOOL ;
    B6 : BOOL ;
    B7 : BOOL ;
   END_STRUCT ;
   L3 : STRUCT
    B8 : BOOL ;
    B9 : BOOL ;
    B10 : BOOL ;
    B11 : BOOL ;
    B12 : BOOL ;
    B13 : BOOL ;
    B14 : BOOL ;
    B15 : BOOL ;
    B0 : BOOL ;
    B1 : BOOL ;
    B2 : BOOL ;
    B3 : BOOL ;
    B4 : BOOL ;
    B5 : BOOL ;
    B6 : BOOL ;
    B7 : BOOL ;
   END_STRUCT ;
   L4 : STRUCT
    B8 : BOOL ;
    B9 : BOOL ;
    B10 : BOOL ;
    B11 : BOOL ;
    B12 : BOOL ;
    B13 : BOOL ;
    B14 : BOOL ;
    B15 : BOOL ;
    B0 : BOOL ;
    B1 : BOOL ;
    B2 : BOOL ;
    B3 : BOOL ;
    B4 : BOOL ;
    B5 : BOOL ;
    B6 : BOOL ;
    B7 : BOOL ;
   END_STRUCT ;
   L5 : STRUCT
    B8 : BOOL ;
    B9 : BOOL ;
    B10 : BOOL ;
    B11 : BOOL ;
    B12 : BOOL ;
    B13 : BOOL ;
    B14 : BOOL ;
    B15 : BOOL ;
    B0 : BOOL ;
    B1 : BOOL ;
    B2 : BOOL ;
    B3 : BOOL ;
    B4 : BOOL ;
    B5 : BOOL ;
    B6 : BOOL ;
    B7 : BOOL ;
   END_STRUCT ;
   L6 : STRUCT
    B8 : BOOL ;
    B9 : BOOL ;
    B10 : BOOL ;
    B11 : BOOL ;
    B12 : BOOL ;
    B13 : BOOL ;
    B14 : BOOL ;
    B15 : BOOL ;
    B0 : BOOL ;
    B1 : BOOL ;
    B2 : BOOL ;
    B3 : BOOL ;
    B4 : BOOL ;
    B5 : BOOL ;
    B6 : BOOL ;
    B7 : BOOL ;
   END_STRUCT ;
   L7 : STRUCT
    B8 : BOOL ;
    B9 : BOOL ;
    B10 : BOOL ;
    B11 : BOOL ;
    B12 : BOOL ;
    B13 : BOOL ;
    B14 : BOOL ;
    B15 : BOOL ;
    B0 : BOOL ;
    B1 : BOOL ;
    B2 : BOOL ;
    B3 : BOOL ;
    B4 : BOOL ;
    B5 : BOOL ;
    B6 : BOOL ;
    B7 : BOOL ;
   END_STRUCT ;
   L8 : STRUCT
    B8 : BOOL ;
    B9 : BOOL ;
    B10 : BOOL ;
    B11 : BOOL ;
    B12 : BOOL ;
    B13 : BOOL ;
    B14 : BOOL ;
    B15 : BOOL ;
    B0 : BOOL ;
    B1 : BOOL ;
    B2 : BOOL ;
    B3 : BOOL ;
    B4 : BOOL ;
    B5 : BOOL ;
    B6 : BOOL ;
    B7 : BOOL ;
   END_STRUCT ;
   L9 : STRUCT
    B8 : BOOL ;
    B9 : BOOL ;
    B10 : BOOL ;
    B11 : BOOL ;
    B12 : BOOL ;
    B13 : BOOL ;
    B14 : BOOL ;
    B15 : BOOL ;
    B0 : BOOL ;
    B1 : BOOL ;
    B2 : BOOL ;
    B3 : BOOL ;
    B4 : BOOL ;
    B5 : BOOL ;
    B6 : BOOL ;
    B7 : BOOL ;
   END_STRUCT ;
  END_STRUCT ;	
END_TYPE

TYPE "ASW_UserSectionState"	// UDT 1002
VERSION : 0.0
  STRUCT
   stEmptying : BOOL ;
   stEmptied : BOOL ;
   stIdling : BOOL ;
   stFault : BOOL ;
   stHand : BOOL ;
   stHold : BOOL ;
   stStep : BOOL ;
   spare : BOOL ;
   stPassive : BOOL ;
   stWait : BOOL ;
   stStarting : BOOL ;
   stStarted : BOOL ;
   stStopping : BOOL ;
   stStopped : BOOL ;
   stFeeding : BOOL ;
   stReady : BOOL ;
  END_STRUCT ;	
END_TYPE

TYPE "ASW_ProductInfo"	// UDT 1003
VERSION : 0.1
  STRUCT
   ProductIdent : STRING  [16 ] := 'ABCDEFGHIJKLMNOP';
   ProductName : STRING  [32 ] := 'ABCDEFGHIJKLMNOPQRSTUVWXYZ012345';
   LOT_NR_1 : STRING  [16 ] := 'ABCDEFGHIJKLMNOP';
   LOT_NR_2 : STRING  [16 ] := 'ABCDEFGHIJKLMNOP';
   LOT_NR_3 : STRING  [16 ] := 'ABCDEFGHIJKLMNOP';
   Reserve : ARRAY  [106 .. 149 ] OF BYTE ;
  END_STRUCT ;	
END_TYPE

TYPE "ASW_HandAddInfo"	// UDT 1004
VERSION : 0.1
  STRUCT
   HandAddNr : INT ;
   ProductIdent : STRING  [16 ] := 'ABCDEFGHIJKLMNOP';
   ProductName : STRING  [32 ] := 'ABCDEFGHIJKLMNOPQRSTUVWXYZ012345';
   Barcode : STRING  [32 ] := 'ABCDEFGHIJKLMNOPQRSTUVWXYZ012345';
   TargetWeight : DINT ;	//Target Weight [gr]
   Reserve : ARRAY  [92 .. 99 ] OF BYTE ;
  END_STRUCT ;	
END_TYPE

TYPE "ASW_DFCARecipe"	// UDT 1005
VERSION : 0.0
  STRUCT
   DFCx : STRUCT 	//Pressensteuerung DFCA/DFCB/DFBB
    maxCurrentPelletmill : INT ;	//max. Pressenstrom [0..599]A
    maxDosingSpeed : INT ;	//max.Dosierdrehzahl Standard [0..100]%
    maxDosingSpeed_2 : INT ;	//MU: max.Dosierdrehzahl Stufe 2  [0..100]%
    maxDosingSpeed_3 : INT ;	//MU: max.Dosierdrehzahl Stufe 3  [0..100]%
    maxConditTemp : INT ;	//max.KonditionierTemp.  [0..100]°C
    nomValLiq_1_Melasse : INT ;	//Sollwert Flüssigkeit 1 [0..200]%o
    nomValLiq_2_Reserve : INT ;	//Sollwert Flüssigkeit 2 [0..200]%o
    nomValLiq_3_Reserve : INT ;	//DFCA: Sollwert Flüssigkeit 3 [0..200]%o
    nomValRollGapAdjust : INT ;	//Sollwert hydr.Rollenverstellung [0..999]x0.1mm
    nomValCoolerOutlet : INT ;	//Sollwert Kühleraustragsleistung [0..100]% (Fein <= 50 / Grob > 50)
    selectPID_ParaSet : INT ;	//Anwahl Regler Parametersatz [1..3]
    nomValRetentionTime : INT ;	//DFBB/DFCB: Sollwert Verweilzeit
    nomValBulkDensity : INT ;	//DFBB/DFCB: spez.Gewicht [100..1000]xkg/m3
    TroughputBy100Proc : DINT ;	//max.Durchsatz bei 100% Drehzahl [0..50000]kg/h
    PelletingDieName : ARRAY  [1 .. 10 ] OF //Form Name
    CHAR ;
    ParameterSetIdent : ARRAY  [1 .. 16 ] OF //Parametersatz Ident (RezeptIdent)
    CHAR ;
    spare56 : INT ;	//---
    spare58 : INT ;	//---
    ParameterSetName : ARRAY  [1 .. 30 ] OF //Parametersatz Name  (Rezeptname)
    CHAR ;
    SPARE_90 : ARRAY  [90 .. 99 ] OF BYTE ;
    optTxtPar1 : STRUCT
     Bit00 : BOOL ;
     Bit01 : BOOL ;
     Bit02 : BOOL ;
    END_STRUCT ;
    optTxtPar2 : STRUCT
     Bit00 : BOOL ;
     Bit01 : BOOL ;
     Bit02 : BOOL ;
    END_STRUCT ;
    optTxtPar3 : STRUCT
     Bit00 : BOOL ;
     Bit01 : BOOL ;
     Bit02 : BOOL ;
    END_STRUCT ;
    optTxtPar4 : STRUCT
     Bit00 : BOOL ;
     Bit01 : BOOL ;
     Bit02 : BOOL ;
    END_STRUCT ;
    optTxtPar5 : STRUCT
     Bit00 : BOOL ;
     Bit01 : BOOL ;
     Bit02 : BOOL ;
    END_STRUCT ;
    optTxtPar6 : STRUCT
     Bit00 : BOOL ;
     Bit01 : BOOL ;
     Bit02 : BOOL ;
    END_STRUCT ;
    optTxtPar7 : STRUCT
     Bit00 : BOOL ;
     Bit01 : BOOL ;
     Bit02 : BOOL ;
    END_STRUCT ;
    optTxtPar8 : STRUCT
     Bit00 : BOOL ;
     Bit01 : BOOL ;
     Bit02 : BOOL ;
    END_STRUCT ;
    optTxtPar9 : STRUCT
     Bit00 : BOOL ;
     Bit01 : BOOL ;
     Bit02 : BOOL ;
    END_STRUCT ;
    optTxtPar10 : STRUCT
     Bit00 : BOOL ;
     Bit01 : BOOL ;
     Bit02 : BOOL ;
    END_STRUCT ;
    optNumPar1 : WORD ;
    optNumPar2 : WORD ;
    optNumPar3 : WORD ;
    optNumPar4 : WORD ;
    optNumPar5 : WORD ;
    optNumPar6 : WORD ;
    optNumPar7 : WORD ;
    optNumPar8 : WORD ;
    optNumPar9 : WORD ;
    optNumPar10 : WORD ;
   END_STRUCT ;
   SPARE_140 : ARRAY  [140 .. 159 ] OF BYTE ;
   PPA : STRUCT 	//SPARE: Post Pelleting Application
    nomValLiquid_1 : INT ;	//Sollwert PPA Flüssigkeit 1 [0..200]%o
    nomValLiquid_2 : INT ;	//Sollwert PPA Flüssigkeit 2 [0..200]%o
    nomValLiquid_3 : INT ;	//Sollwert PPA Flüssigkeit 3 [0..200]%o
    nomValLiquid_4 : INT ;	//Sollwert PPA Flüssigkeit 4 [0..200]%o
    nomValLiquid_5 : INT ;	//Sollwert PPA Flüssigkeit 5 [0..200]%o
    nomValLiquid_6 : INT ;	//Sollwert PPA Flüssigkeit 6 [0..200]%o
    nomValLiquid_7 : INT ;	//Sollwert PPA Flüssigkeit 7 [0..200]%o
    nomValLiquid_8 : INT ;	//Sollwert PPA Flüssigkeit 8 [0..200]%o
    nomValLiquid_9 : INT ;	//Sollwert PPA Flüssigkeit 9 [0..200]%o
    nomValLiquid_10 : INT ;	//Sollwert PPA Flüssigkeit 10 [0..200]%o
    nomValLiquid_11 : INT ;	//Sollwert PPA Flüssigkeit 11 [0..200]%o
    nomValLiquid_12 : INT ;	//Sollwert PPA Flüssigkeit 12 [0..200]%o
   END_STRUCT ;
   SPARE_184 : ARRAY  [184 .. 199 ] OF BYTE ;
  END_STRUCT ;	
END_TYPE

TYPE "GCS7_UDT_FunctionKey"	// UDT 10601
VERSION : 0.0
  STRUCT
   CmdProdCheck : BOOL ;	//ASW: Start after product check
   CmdEmptying : BOOL ;
   CmdTolerate : BOOL ;
   CmdHornOff : BOOL ;
   Cmd04 : BOOL ;
   Cmd05 : BOOL ;
   Cmd06 : BOOL ;
   Cmd07 : BOOL ;
   CmdStart : BOOL ;
   CmdTransferOn : BOOL ;
   CmdFeedOn : BOOL ;
   CmdFree : BOOL ;
   CmdAutomatic : BOOL ;
   CmdStepOff : BOOL ;
   CmdNextStep : BOOL ;
   CmdAcceptSize : BOOL ;
   Cmd16 : BOOL ;
   CmdAbortBatch : BOOL ;
   CmdFaultReset : BOOL ;
   CmdHornOn : BOOL ;
   Cmd17 : BOOL ;
   Cmd18 : BOOL ;
   Cmd19 : BOOL ;
   CmdHLOverride : BOOL ;	//ASW: Activate function override HL
   CmdImmediateStop : BOOL ;
   CmdTransferOff : BOOL ;
   CmdFeedOff : BOOL ;
   CmdHold : BOOL ;
   CmdHand : BOOL ;
   CmdStepOn : BOOL ;
   CmdReset : BOOL ;
   CmdSequenzStop : BOOL ;
  END_STRUCT ;	
END_TYPE

TYPE "GCS7_UDT_FaultPattern"	// UDT 10602
VERSION : 0.0
  STRUCT
   Es00 : BOOL ;
   Es01 : BOOL ;
   Es02 : BOOL ;
   Es03 : BOOL ;
   Es04 : BOOL ;
   Es05 : BOOL ;
   Es06 : BOOL ;
   Es07 : BOOL ;
   Es08 : BOOL ;
   Es09 : BOOL ;
   Es10 : BOOL ;
   Es11 : BOOL ;
   Es12 : BOOL ;
   Es13 : BOOL ;
   Es14 : BOOL ;
   EsNewBinTimeout : BOOL ;	//ASW: Max. delay time to send a new bin
   EsBatchSize : BOOL ;
   EsRefillLevel : BOOL ;
   EsSectionTimeOut : BOOL ;	//ASW: Max. section time to stay in section
   EsHandAddTimeOut : BOOL ;	//ASW: Max. delay time to accept manual ingredients
   EsRecipePlace : BOOL ;	//ASW: Fault recipe place
   EsProductMismatch : BOOL ;	//ASW: Product check failed
   Es22 : BOOL ;
   Es23 : BOOL ;
   EsEmpty : BOOL ;
   EsFull : BOOL ;
   EsWayConflict : BOOL ;
   EsWarning : BOOL ;
   EsMech : BOOL ;
   EsDosing : BOOL ;
   EsEmptying : BOOL ;
   EsInterrupt : BOOL ;
  END_STRUCT ;	
END_TYPE

TYPE "GCS7_UDT_StatusPattern"	// UDT 10603
VERSION : 0.0
  STRUCT
   StaStartRelease : BOOL ;
   StaMixingTime : BOOL ;
   StaMixingTimeEnd : BOOL ;
   Sta03 : BOOL ;
   Sta04 : BOOL ;
   Sta05 : BOOL ;
   Sta06 : BOOL ;
   StaDPFault : BOOL ;
   StaHWStop : BOOL ;
   StaAutostartSec : BOOL ;
   StaAutostart : BOOL ;
   StaOnline : BOOL ;
   StaLoaded : BOOL ;
   StaHandAdd : BOOL ;
   StaEmptyingTime : BOOL ;
   StaStartwarning : BOOL ;
   StaImmediateStopASW : BOOL ;	//ASW: Summary information: Any condition is true
   StaTransferOffASW : BOOL ;	//ASW: Summary information: Any condition is true
   StaFeedOffASW : BOOL ;	//ASW: Summary information: Any condition is true
   Sta23 : BOOL ;
   Sta24 : BOOL ;
   Sta25 : BOOL ;
   Sta26 : BOOL ;
   StaHLOverride : BOOL ;	//ASW: Override function is active
   StaImmediateStop : BOOL ;
   StaTransferOff : BOOL ;
   StaFeedOff : BOOL ;
   StaHold : BOOL ;
   StaHand : BOOL ;
   StaStep : BOOL ;
   StaReset : BOOL ;
   StaEndOfJob : BOOL ;
  END_STRUCT ;	
END_TYPE

TYPE "MELEYieldScale"	// UDT 19000
VERSION : 0.1
  STRUCT
   PCCScaleNo : DINT ;
   ActualFlowrate : DINT ;
   ActualJobWeight : DINT ;
   NonEraseableWeight : DINT ;
  END_STRUCT ;	
END_TYPE

TYPE "WinCoSYieldScale"	// UDT 19001
VERSION : 0.1
  STRUCT
   PCCScaleNo : DINT ;
   JobIdent : DINT ;
   ActualFlowrate : DINT ;
   ActualJobWeight : DINT ;
   NonEraseableWeight : DINT ;
  END_STRUCT ;	
END_TYPE

TYPE "SamplerData"	// UDT 19002
VERSION : 0.1
  STRUCT
   F_Result : ARRAY  [1 .. 16 ] OF BOOL ;
   Sampler : ARRAY  [1 .. 1 ] OF STRUCT
    Number : INT ;
    BottleID : DINT ;
    NoOfSamples : INT ;
    SampleTime : INT ;
    JobID : DINT ;
   END_STRUCT ;
  END_STRUCT ;	
END_TYPE

TYPE "BigBagData"	// UDT 19003
VERSION : 0.1
  STRUCT
   F_Result : ARRAY  [1 .. 16 ] OF BOOL ;
   BigBag : ARRAY  [1 .. 1 ] OF
   STRUCT
    Number : INT ;
    Weight : DINT ;	//gr
    Days : INT ;	//Days from 01.01.1990
    Minutes : INT ;	//Minutes of the day
    Seconds : INT ;	//Seconds
    JobID : DINT ;
   END_STRUCT ;
  END_STRUCT ;	
END_TYPE

TYPE "GCS7_FB9_Communication"	// UDT 20099
VERSION : 0.1
  STRUCT
   StStopped : BOOL ;	//to virtual group
   StStarting : BOOL ;	//to virtual group
   StStarted : BOOL ;	//to virtual group
   StStopping : BOOL ;	//to virtual group
   StFault : BOOL ;	//to virtual group
   OutWarning : BOOL ;	//to virtual group
   InManual : BOOL ;	//to virtual group
   InHWStop : BOOL ;	//to virtual group
   InDPFault : BOOL ;	//to virtual group
   InLoaded : BOOL ;	//to virtual group
   InAutoStart : BOOL ;	//to virtual group
   InStartWarning : BOOL ;	//to virtual group
   ASW14 : BOOL ;	//to virtual group
   ASW15 : BOOL ;	//to virtual group
   SelectedForPLC1 : BOOL ;	//to virtual group
   SelectedForPLC2 : BOOL ;	//to virtual group
   SelectedForPLC3 : BOOL ;	//to virtual group
   SelectedForPLC4 : BOOL ;	//to virtual group
   MultipleUsed : BOOL ;	//to virtual group
   SelectedForPLC5 : BOOL ;	//to virtual group
   SelectedForPLC6 : BOOL ;	//to virtual group
   StCode : INT ;	//to virtual group
   InEnableGr : BOOL ;	//to real group
   spare11 : BOOL ;	//to real group
   CmdNext : BOOL ;	//to real group
   CmdFaultReset : BOOL ;	//to real group
   InOccupied : BOOL ;	//to real group
   CmdManualOff : BOOL ;	//to real group
   CmdNewJob : BOOL ;	//to real group
   CmdNewValue : BOOL ;	//to real group
   CmdRestartIdling : BOOL ;	//to real group
   CmdContinue : BOOL ;	//to real group
   ASW32 : BOOL ;	//to real group
   ASW33 : BOOL ;	//to real group
   ASW34 : BOOL ;	//to real group
   ASW35 : BOOL ;	//to real group
   InClose : BOOL ;	//to real group
   InOpen : BOOL ;	//to real group
  END_STRUCT ;	
END_TYPE

